// TIA Portal V16 program export: 0 tag tables, 0 data types, 18 data blocks, 36 code blocks (in call order from the OBs), 5 instance data blocks

DATA_BLOCK "dbAlarms"   // DB106
{ S7_Optimized_Access := 'FALSE'; DB_Accessible_From_OPC_UA := 'FALSE' }
VERSION : 0.1
// stored: AutoNumber false, DBAccessibleFromOPCUA false, IsOnlyStoredInLoadMemory false, IsWriteProtectedInAS false
   VAR
      PLI : Array[1..4, 1..32] of Bool;
   END_VAR
BEGIN
   PLI[1,1..32] := FALSE;
   PLI[2,1..32] := FALSE;
   PLI[3,1..32] := FALSE;
   PLI[4,1..32] := FALSE;
END_DATA_BLOCK

DATA_BLOCK "dbDI"   // DB10
{ S7_Optimized_Access := 'FALSE'; DB_Accessible_From_OPC_UA := 'FALSE' }
VERSION : 0.1
// stored: AutoNumber false, DBAccessibleFromOPCUA false, IsOnlyStoredInLoadMemory false, IsWriteProtectedInAS false
   VAR
      ZAUSTAVITEV_V_SILI_NI_AKTIVIRANA : Bool;   // 0=NOT OK, 1=OK
      FOTO_ZAVESA_KANAL_1 : Bool;   // 0=NOT OK, 1=OK
      FOTO_ZAVESA_KANAL_2 : Bool;   // 0=NOT OK, 1=OK
      START_LEVO_NA_VPENJANJU : Bool;
      START_DESNO_NA_VPENJANJU : Bool;
      Spare0_5 : Bool;
      Spare0_6 : Bool;
      PRISOTNOST_ZRAKA_NA_NAPRAVI : Bool;   // 0=NOT OK, 1=OK
      Spare1_0 : Bool;
      Spare1_1 : Bool;
      Spare1_2 : Bool;
      Spare1_3 : Bool;
      Spare1_4 : Bool;
      Spare1_5 : Bool;
      Spare1_6 : Bool;
      Spare1_7 : Bool;
      BIMETAL_TRANSPORTA_NOGIC_IZKLJUCIL : Bool;   // (I0.0) / 0=NOT OK, 1=OK
      VIBRATOR_NOGIC_READY : Bool;   // (I0.1) / 0=NOT READY, 1=READY
      BIMETAL_VIJACENJA_NOGIC_IZKLJUCIL : Bool;   // (I0.2) / 0=NOT OK, 1=OK
      FR_MOTORJA1_ZADAJ_DESNO_READY : Bool;   // (I0.3) / 0=NOT READY, 1=READY
      FR_MOTORJA2_SPREDAJ_DESNO_READY : Bool;   // (I0.4) / 0=NOT READY, 1=READY
      FR_MOTORJA1_ZADAJ_LEVO_READY : Bool;   // (I0.5) / 0=NOT READY, 1=READY
      FR_MOTORJA2_SPREDAJ_LEVO_READY : Bool;   // (I0.6) / 0=NOT READY, 1=READY
      Spare20_7 : Bool;
      FOTOCELICA_TRANSPORTA_NOGIC : Bool;   // (I0.7) / 0=NI PRISOTNO, 1=PRISOTNO | NOT USED
      FOTOCELICA_VSTOP_DRCA_NOGIC : Bool;   // (I1.0) / 0=NI PRISOTNO, 1=PRISOTNO | ? | NOT USED
      FOTOCELICA_PRED_MESTOM_LOCEVANJA : Bool;   // (I1.1) / 0=NI PRISOTNO, 1=PRISOTNO | NOT USED
      FOTOCELICA_VSTOP_DRCA_LEVO : Bool;   // (I1.2) / 0=NI PRISOTNO, 1=PRISOTNO | NOT USED
      FOTOCELICA_VSTOP_DRCA_DESNO : Bool;   // (I1.3) / 0=NI PRISOTNO, 1=PRISOTNO | NOT USED
      FOTOCELICA_LOC_IZH_DRCA_LEVO : Bool;   // (I1.4) / 0=NI PRISOTNO, 1=PRISOTNO | NOT USED
      FOTOCELICA_LOC_IZH_DRCA_DESNO : Bool;   // (I1.5) / 0=NI PRISOTNO, 1=PRISOTNO | NOT USED
      NOGICE_V_VIBRATORJU : Bool;
      ROTACIJSKI_CIL_DESNO : Bool;   // 0=NI PRISOTNO, 1=PRISOTNO
      ROTACIJSKI_CIL_SREDINA : Bool;   // 0=NI PRISOTNO, 1=PRISOTNO
      ROTACIJSKI_CIL_LEVO : Bool;   // 0=NI PRISOTNO, 1=PRISOTNO
      LOC_DRCA_DESNO_NAPREJ : Bool;   // 0=NI PRISOTNO, 1=PRISOTNO | NOT USED
      LOC_DRCA_DESNO_NAZAJ : Bool;   // 0=NI PRISOTNO, 1=PRISOTNO | NOT USED
      LOC_DRCA_LEVO_NAZAJ : Bool;   // 0=NI PRISOTNO, 1=PRISOTNO | NOT USED
      LOC_DRCA_LEVO_NAPREJ : Bool;   // 0=NI PRISOTNO, 1=PRISOTNO | NOT USED
      Spare22_7 : Bool;
      FOTOCELICA_LOC_TRAK_DESNO1 : Bool;   // 0=NI PRISOTNO, 1=PRISOTNO | NOT USED
      FOTOCELICA_LOC_TRAK_DESNO2 : Bool;   // 0=NI PRISOTNO, 1=PRISOTNO | NOT USED
      FOTOCELICA_VIJACENJE_DESNOZADAJ : Bool;   // 0=NI PRISOTNO, 1=PRISOTNO | NOT USED
      FOTOCELICA_VIJACENJE_DESNOSPREDAJ : Bool;   // 0=NI PRISOTNO, 1=PRISOTNO | NOT USED
      VIJACENJE_DESNO_1_NAZAJ : Bool;   // LOCEVANJE NA TRAKU DESNO NAZAJ
      VIJACENJE_DESNO_1_NAPREJ : Bool;   // LOCEVANJE NA TRAKU DESNO NAPREJ
      MESTO_VIJAC_STOP_DESNO_ZAD_NAZAJ : Bool;   // 0=NI PRISOTNO, 1=PRISOTNO
      MESTO_VIJAC_STOP_DESNO_ZAD_NAPREJ : Bool;   // 0=NI PRISOTNO, 1=PRISOTNO
      MESTO_VIJACENJE_DESNO_ZAD_DVIG_DOL : Bool;   // (I1.6) / 0=NI PRISOTNO, 1=PRISOTNO | ? Detekcija spodnje lege cilindra spusta| DONE Man
      MESTO_VIJACENJE_DESNO_ZAD_CENT_NARAZEN : Bool;   // (I1.7) / 0=NI PRISOTNO, 1=PRISOTNO
      MESTO_VIJACENJE_DESNO_ZAD_CENT_SKUPAJ : Bool;   // 0=NI PRISOTNO, 1=PRISOTNO
      Spare24_3 : Bool;   // MESTO_VIJACENJE_DESNO_SPRED_NAZAJ "STOP_DESNO_SPRED_NAZAJ(Spare23_4) ne obstaja. Konec traka ne obstaja cilinder za stopanje nogice.
      Spare24_4 : Bool;   // MESTO_VIJACENJE_DESNO_SPRED_NAPREJ "STOP_DESNO_SPRED_NAPREJ (Spare23_5) ne obstaja. Konec traka ne obstaja cilinder za stopanje nogice.
      MESTO_VIJACENJE_DESNO_SPRED_DVIG_DOL : Bool;   // 0=NI PRISOTNO, 1=PRISOTNO | ? Detekcija spodnje lege cilindra spusta| DONE Man
      MESTO_VIJACENJE_DESNO_SPRED_CENT_NARAZEN : Bool;   // 0=NI PRISOTNO, 1=PRISOTNO
      MESTO_VIJACENJE_DESNO_SPRED_CENT_SKUPAJ : Bool;   // 0=NI PRISOTNO, 1=PRISOTNO
      KONCNA_POZICIJA_VIJACENJA_DES_NAZAJ : Bool;   // 0=NI PRISOTNO, 1=PRISOTNO | NOT USED
      KONCNA_POZICIJA_VIJACENJA_DES_NAPREJ : Bool;   // 0=NI PRISOTNO, 1=PRISOTNO | NOT USED
      Spare25_2 : Bool;
      Spare25_3 : Bool;
      KONCNA_POZICIJA_VIJACENJA_LEVO_NAZAJ : Bool;   // 0=NI PRISOTNO, 1=PRISOTNO | NOT USED
      KONCNA_POZICIJA_VIJACENJA_LEVO_NAPREJ : Bool;   // 0=NI PRISOTNO, 1=PRISOTNO | NOT USED
      Spare25_6 : Bool;
      Spare25_7 : Bool;
      FOTOCELICA_LOC_TRAK_LEVO1 : Bool;   // 0=NI PRISOTNO, 1=PRISOTNO | NOT USED
      FOTOCELICA_LOC_TRAK_LEVO2 : Bool;   // 0=NI PRISOTNO, 1=PRISOTNO | NOT USED
      FOTOCELICA_VIJACENJE_LEVO_ZADAJ : Bool;   // 0=NI PRISOTNO, 1=PRISOTNO | NOT USED
      FOTOCELICA_VIJACENJE_LEVO_SPREDAJ : Bool;   // 0=NI PRISOTNO, 1=PRISOTNO | NOT USED
      VIJACENJE_LEVO_1_NAZAJ : Bool;   // LOCEVANJE NA TRAKU LEVO NAZAJ
      VIJACENJE_LEVO_1_NAPREJ : Bool;   // LOCEVANJE NA TRAKU LEVO NAPREJ
      MESTO_VIJAC_STOP_LEVO_ZAD_NAZAJ : Bool;   // 0=NI PRISOTNO, 1=PRISOTNO
      MESTO_VIJAC_STOP_LEVO_ZAD_NAPREJ : Bool;   // 0=NI PRISOTNO, 1=PRISOTNO
      MESTO_VIJACENJE_LEVO_ZAD_DVIG_DOL : Bool;   // 0=NI PRISOTNO, 1=PRISOTNO | ? Detekcija spodnje lege cilindra spusta| DONE Man
      MESTO_VIJACENJE_LEVO_ZAD_CENT_NARAZEN : Bool;   // 0=NI PRISOTNO, 1=PRISOTNO
      MESTO_VIJACENJE_LEVO_ZAD_CENT_SKUPAJ : Bool;   // 0=NI PRISOTNO, 1=PRISOTNO
      Spare27_3 : Bool;   // MESTO_VIJACENJE_LEVO_SPRED_NAZAJ "STOP_LEVO_SPRED_NAZAJ(Spare26_4) ne obstaja. Konec traka ne obstaja cilinder za stopanje nogice.
      Spare27_4 : Bool;   // MESTO_VIJACENJE_LEVO_SPRED_NAPREJ "STOP_LEVO_SPRED_NAPREJ (Spare26_5) ne obstaja. Konec traka ne obstaja cilinder za stopanje nogice.
      MESTO_VIJACENJE_LEVO_SPRED_DVIG_DOL : Bool;   // 0=NI PRISOTNO, 1=PRISOTNO | ? Detekcija spodnje lege cilindra spusta| DONE Man
      MESTO_VIJACENJE_LEVO_SPRED_CENT_NARAZEN : Bool;   // 0=NI PRISOTNO, 1=PRISOTNO
      MESTO_VIJACENJE_LEVO_SPRED_CENT_SKUPAJ : Bool;   // 0=NI PRISOTNO, 1=PRISOTNO
      INDUKTIVEC_PRAVILNA_VLOZITEV_DNA_1 : Bool;   // 0=NI PRISOTNO, 1=PRISOTNO | NOT USED
      INDUKTIVEC_PRAVILNA_VLOZITEV_DNA_2 : Bool;   // 0=NI PRISOTNO, 1=PRISOTNO | NOT USED
      VPENJANJE_DNA_LEVO_ZADAJ_GOR : Bool;   // 0=NI PRISOTNO, 1=PRISOTNO
      VPENJANJE_DNA_LEVO_ZADAJ_DOL : Bool;   // 0=NI PRISOTNO, 1=PRISOTNO
      VPENJANJE_DNA_LEVO_SPREDAJ_GOR : Bool;   // 0=NI PRISOTNO, 1=PRISOTNO
      VPENJANJE_DNA_LEVO_SPREDAJ_DOL : Bool;   // 0=NI PRISOTNO, 1=PRISOTNO
      VPENJANJE_DNA_DESNO_ZADAJ_GOR : Bool;   // 0=NI PRISOTNO, 1=PRISOTNO
      VPENJANJE_DNA_DESNO_ZADAJ_DOL : Bool;   // 0=NI PRISOTNO, 1=PRISOTNO
      VPENJANJE_DNA_DESNO_SPREDAJ_GOR : Bool;   // 0=NI PRISOTNO, 1=PRISOTNO
      VPENJANJE_DNA_DESNO_SPREDAJ_DOL : Bool;   // 0=NI PRISOTNO, 1=PRISOTNO
      Static_1 : Bool;   // 0=NI PRISOTNO, 1=PRISOTNO
      Spare29_3 : Bool;
      Spare29_4 : Bool;
      Spare29_5 : Bool;
      Spare29_6 : Bool;
      Spare29_7 : Bool;
   END_VAR
BEGIN
END_DATA_BLOCK

DATA_BLOCK "dbDO"   // DB11
{ S7_Optimized_Access := 'FALSE'; DB_Accessible_From_OPC_UA := 'FALSE' }
VERSION : 0.1
// stored: AutoNumber false, DBAccessibleFromOPCUA false, IsOnlyStoredInLoadMemory false, IsWriteProtectedInAS false
   VAR
      SEMAFOR_ZELENA : Bool;
      SEMAFOR_RUMENA : Bool;
      SEMAFOR_RDECA : Bool;
      Spare0_3 { ExternalAccessible := 'False'; ExternalVisible := 'False'; ExternalWritable := 'False'} : Bool;
      Spare0_4 { ExternalAccessible := 'False'; ExternalVisible := 'False'; ExternalWritable := 'False'} : Bool;
      Spare0_5 { ExternalAccessible := 'False'; ExternalVisible := 'False'; ExternalWritable := 'False'} : Bool;
      Spare0_6 { ExternalAccessible := 'False'; ExternalVisible := 'False'; ExternalWritable := 'False'} : Bool;
      Spare0_7 { ExternalAccessible := 'False'; ExternalVisible := 'False'; ExternalWritable := 'False'} : Bool;
      Spare1_0 { ExternalAccessible := 'False'; ExternalVisible := 'False'; ExternalWritable := 'False'} : Bool;
      Spare1_1 { ExternalAccessible := 'False'; ExternalVisible := 'False'; ExternalWritable := 'False'} : Bool;
      Spare1_2 { ExternalAccessible := 'False'; ExternalVisible := 'False'; ExternalWritable := 'False'} : Bool;
      Spare1_3 { ExternalAccessible := 'False'; ExternalVisible := 'False'; ExternalWritable := 'False'} : Bool;
      Spare1_4 { ExternalAccessible := 'False'; ExternalVisible := 'False'; ExternalWritable := 'False'} : Bool;
      Spare1_5 { ExternalAccessible := 'False'; ExternalVisible := 'False'; ExternalWritable := 'False'} : Bool;
      Spare1_6 { ExternalAccessible := 'False'; ExternalVisible := 'False'; ExternalWritable := 'False'} : Bool;
      Spare1_7 { ExternalAccessible := 'False'; ExternalVisible := 'False'; ExternalWritable := 'False'} : Bool;
      VKLOP_M_TRACNEGA_TRANS_NOGIC : Bool;   // (Q0.0)
      VKLOP_VIBRATORJA : Bool;   // (Q0.1)
      VKLOP_M_TRAKA_VIJACNIKA : Bool;   // (Q0.2)
      Spare20_3 { ExternalAccessible := 'False'; ExternalVisible := 'False'; ExternalWritable := 'False'} : Bool;
      Spare20_4 { ExternalAccessible := 'False'; ExternalVisible := 'False'; ExternalWritable := 'False'} : Bool;
      Spare20_5 { ExternalAccessible := 'False'; ExternalVisible := 'False'; ExternalWritable := 'False'} : Bool;
      Spare20_6 { ExternalAccessible := 'False'; ExternalVisible := 'False'; ExternalWritable := 'False'} : Bool;
      Spare20_7 { ExternalAccessible := 'False'; ExternalVisible := 'False'; ExternalWritable := 'False'} : Bool;
      MOTOR_1_ZADAJ_DESNO_START : Bool;   // (Q1.1)
      MOTOR_1_ZADAJ_DESNO_RESET : Bool;   // (Q1.2)
      MOTOR_1_ZADAJ_DESNO_HITROST : Bool;   // (Q1.3)
      MOTOR_1_ZADAJ_DESNO_SMER : Bool;   // (Q1.4)
      MOTOR_2_SPREDAJ_DESNO_START : Bool;   // (Q1.5)
      MOTOR_2_SPREDAJ_DESNO_RESET : Bool;   // (Q1.6)
      MOTOR_2_SPREDAJ_DESNO_HITROST : Bool;   // (Q1.7)
      MOTOR_2_SPREDAJ_DESNO_SMER : Bool;
      MOTOR_1_ZADAJ_LEVO_START : Bool;
      MOTOR_1_ZADAJ_LEVO_RESET : Bool;
      MOTOR_1_ZADAJ_LEVO_HITROST : Bool;
      MOTOR_1_ZADAJ_LEVO_SMER : Bool;
      MOTOR_2_SPREDAJ_LEVO_START : Bool;
      MOTOR_2_SPREDAJ_LEVO_RESET : Bool;
      MOTOR_2_SPREDAJ_LEVO_HITROST : Bool;
      MOTOR_2_SPREDAJ_LEVO_SMER : Bool;
      Spare23_0 { ExternalAccessible := 'False'; ExternalVisible := 'False'; ExternalWritable := 'False'} : Bool;
      Spare23_1 { ExternalAccessible := 'False'; ExternalVisible := 'False'; ExternalWritable := 'False'} : Bool;
      Spare23_2 { ExternalAccessible := 'False'; ExternalVisible := 'False'; ExternalWritable := 'False'} : Bool;
      Spare23_3 { ExternalAccessible := 'False'; ExternalVisible := 'False'; ExternalWritable := 'False'} : Bool;
      Spare23_4 { ExternalAccessible := 'False'; ExternalVisible := 'False'; ExternalWritable := 'False'} : Bool;
      Spare23_5 { ExternalAccessible := 'False'; ExternalVisible := 'False'; ExternalWritable := 'False'} : Bool;
      Spare23_6 { ExternalAccessible := 'False'; ExternalVisible := 'False'; ExternalWritable := 'False'} : Bool;
      Spare23_7 { ExternalAccessible := 'False'; ExternalVisible := 'False'; ExternalWritable := 'False'} : Bool;
   END_VAR
BEGIN
END_DATA_BLOCK

DATA_BLOCK "dbDigitalSensors"   // DB30
{ S7_Optimized_Access := 'FALSE'; DB_Accessible_From_OPC_UA := 'FALSE' }
VERSION : 0.1
// stored: AutoNumber false, DBAccessibleFromOPCUA false, IsOnlyStoredInLoadMemory false, IsWriteProtectedInAS false
   VAR
      ZAUSTAVITEV_V_SILI_NI_AKTIVIRANA : "udtDigitalSensor";
      FOTO_ZAVESA_KANAL_1 : "udtDigitalSensor";
      FOTO_ZAVESA_KANAL_2 : "udtDigitalSensor";
      START_LEVO_NA_VPENJANJU : "udtDigitalSensor";
      START_DESNO_NA_VPENJANJU : "udtDigitalSensor";
      PRISOTNOST_ZRAKA_NA_NAPRAVI : "udtDigitalSensor";
      BIMETAL_TRANSPORTA_NOGIC_IZKLJUCIL : "udtDigitalSensor";
      VIBRATOR_NOGIC_READY : "udtDigitalSensor";
      BIMETAL_VIJACENJA_NOGIC_IZKLJUCIL : "udtDigitalSensor";
      FR_MOTORJA1_ZADAJ_DESNO_READY : "udtDigitalSensor";
      FR_MOTORJA2_SPREDAJ_DESNO_READY : "udtDigitalSensor";
      FR_MOTORJA1_ZADAJ_LEVO_READY : "udtDigitalSensor";
      FR_MOTORJA2_SPREDAJ_LEVO_READY : "udtDigitalSensor";
      Spare20_7 : "udtDigitalSensor";
      FOTOCELICA_TRANSPORTA_NOGIC : "udtDigitalSensor";
      FOTOCELICA_VSTOP_DRCA_NOGIC : "udtDigitalSensor";
      FOTOCELICA_PRED_MESTOM_LOCEVANJA : "udtDigitalSensor";
      FOTOCELICA_VSTOP_DRCA_LEVO : "udtDigitalSensor";
      FOTOCELICA_VSTOP_DRCA_DESNO : "udtDigitalSensor";
      FOTOCELICA_LOC_IZH_DRCA_LEVO : "udtDigitalSensor";
      FOTOCELICA_LOC_IZH_DRCA_DESNO : "udtDigitalSensor";
      NOGICE_V_VIBRATORJU : "udtDigitalSensor";
      ROTACIJSKI_CIL_DESNO : "udtDigitalSensor";
      ROTACIJSKI_CIL_SREDINA : "udtDigitalSensor";
      ROTACIJSKI_CIL_LEVO : "udtDigitalSensor";
      LOC_DRCA_DESNO_NAPREJ : "udtDigitalSensor";
      LOC_DRCA_DESNO_NAZAJ : "udtDigitalSensor";
      LOC_DRCA_LEVO_NAZAJ : "udtDigitalSensor";
      LOC_DRCA_LEVO_NAPREJ : "udtDigitalSensor";
      Spare22_7 : "udtDigitalSensor";
      FOTOCELICA_LOC_TRAK_DESNO1 : "udtDigitalSensor";
      FOTOCELICA_LOC_TRAK_DESNO2 : "udtDigitalSensor";
      FOTOCELICA_VIJACENJE_DESNOZADAJ : "udtDigitalSensor";
      FOTOCELICA_VIJACENJE_DESNOSPREDAJ : "udtDigitalSensor";
      VIJACENJE_DESNO_1_NAZAJ : "udtDigitalSensor";
      VIJACENJE_DESNO_1_NAPREJ : "udtDigitalSensor";
      MESTO_VIJAC_STOP_DESNO_ZAD_NAZAJ : "udtDigitalSensor";
      MESTO_VIJAC_STOP_DESNO_ZAD_NAPREJ : "udtDigitalSensor";
      MESTO_VIJACENJE_DESNO_ZAD_DVIG_DOL : "udtDigitalSensor";
      MESTO_VIJACENJE_DESNO_ZAD_CENT_NARAZEN : "udtDigitalSensor";
      MESTO_VIJACENJE_DESNO_ZAD_CENT_SKUPAJ : "udtDigitalSensor";
      Spare24_3 : "udtDigitalSensor";
      Spare24_4 : "udtDigitalSensor";
      MESTO_VIJACENJE_DESNO_SPRED_DVIG_DOL : "udtDigitalSensor";
      MESTO_VIJACENJE_DESNO_SPRED_CENT_NARAZEN : "udtDigitalSensor";
      MESTO_VIJACENJE_DESNO_SPRED_CENT_SKUPAJ : "udtDigitalSensor";
      KONCNA_POZICIJA_VIJACENJA_DES_NAZAJ : "udtDigitalSensor";
      KONCNA_POZICIJA_VIJACENJA_DES_NAPREJ : "udtDigitalSensor";
      Spare25_2 : "udtDigitalSensor";
      Spare25_3 : "udtDigitalSensor";
      KONCNA_POZICIJA_VIJACENJA_LEVO_NAZAJ : "udtDigitalSensor";
      KONCNA_POZICIJA_VIJACENJA_LEVO_NAPREJ : "udtDigitalSensor";
      Spare25_6 : "udtDigitalSensor";
      Spare25_7 : "udtDigitalSensor";
      FOTOCELICA_LOC_TRAK_LEVO1 : "udtDigitalSensor";
      FOTOCELICA_LOC_TRAK_LEVO2 : "udtDigitalSensor";
      FOTOCELICA_VIJACENJE_LEVO_ZADAJ : "udtDigitalSensor";
      FOTOCELICA_VIJACENJE_LEVO_SPREDAJ : "udtDigitalSensor";
      VIJACENJE_LEVO_1_NAZAJ : "udtDigitalSensor";
      VIJACENJE_LEVO_1_NAPREJ : "udtDigitalSensor";
      MESTO_VIJAC_STOP_LEVO_ZAD_NAZAJ : "udtDigitalSensor";
      MESTO_VIJAC_STOP_LEVO_ZAD_NAPREJ : "udtDigitalSensor";
      MESTO_VIJACENJE_LEVO_ZAD_DVIG_DOL : "udtDigitalSensor";
      MESTO_VIJACENJE_LEVO_ZAD_CENT_NARAZEN : "udtDigitalSensor";
      MESTO_VIJACENJE_LEVO_ZAD_CENT_SKUPAJ : "udtDigitalSensor";
      Spare27_3 : "udtDigitalSensor";
      Spare27_4 : "udtDigitalSensor";
      MESTO_VIJACENJE_LEVO_SPRED_DVIG_DOL : "udtDigitalSensor";
      MESTO_VIJACENJE_LEVO_SPRED_CENT_NARAZEN : "udtDigitalSensor";
      MESTO_VIJACENJE_LEVO_SPRED_CENT_SKUPAJ : "udtDigitalSensor";
      INDUKTIVEC_PRAVILNA_VLOZITEV_DNA_1 : "udtDigitalSensor";
      INDUKTIVEC_PRAVILNA_VLOZITEV_DNA_2 : "udtDigitalSensor";
      VPENJANJE_DNA_LEVO_ZADAJ_GOR : "udtDigitalSensor";
      VPENJANJE_DNA_LEVO_ZADAJ_DOL : "udtDigitalSensor";
      VPENJANJE_DNA_LEVO_SPREDAJ_GOR : "udtDigitalSensor";
      VPENJANJE_DNA_LEVO_SPREDAJ_DOL : "udtDigitalSensor";
      VPENJANJE_DNA_DESNO_ZADAJ_GOR : "udtDigitalSensor";
      VPENJANJE_DNA_DESNO_ZADAJ_DOL : "udtDigitalSensor";
      VPENJANJE_DNA_DESNO_SPREDAJ_GOR : "udtDigitalSensor";
      VPENJANJE_DNA_DESNO_SPREDAJ_DOL : "udtDigitalSensor";
   END_VAR
BEGIN
END_DATA_BLOCK

DATA_BLOCK "dbDigitalValves"   // DB32
{ S7_Optimized_Access := 'FALSE'; DB_Accessible_From_OPC_UA := 'FALSE' }
VERSION : 0.1
// stored: AutoNumber false, DBAccessibleFromOPCUA false, IsOnlyStoredInLoadMemory false, IsWriteProtectedInAS false
   VAR
      Y17_RotCilipozDesno : "udtDigitalValve";   // Crane control not selected lamps (Q0.0)
      Y18_RotCilipozLevo : "udtDigitalValve";
      Y2_VijaDesZad_Dvig : "udtDigitalValve";
      Y3_VijaDesSpr_Dvig : "udtDigitalValve";
      Y4_VijaLevZad_Dvig : "udtDigitalValve";
      Y5_VijaLevSpr_Dvig : "udtDigitalValve";
      Y6_DrcaLocev_Des : "udtDigitalValve";
      Y7_DrcaLocev_Lev : "udtDigitalValve";
      Y8_VijaLocev_Des : "udtDigitalValve";
      Y9_VijaStop_DesZad : "udtDigitalValve";
      Y10_Centri_DesZad : "udtDigitalValve";
      Y11_Centri_DesSpr : "udtDigitalValve";
      Y12_VijaLocev_Lev : "udtDigitalValve";
      Y13_VijaStop_LevZad : "udtDigitalValve";
      Y14_Centri_LevZad : "udtDigitalValve";
      Y15_Centri_LevSpr : "udtDigitalValve";
      Y16_VpenjanjeDna : "udtDigitalValve";
      SEMAFOR_ZELENA : "udtDigitalValve";
      SEMAFOR_RUMENA : "udtDigitalValve";
      SEMAFOR_RDECA : "udtDigitalValve";
   END_VAR
BEGIN
END_DATA_BLOCK

DATA_BLOCK "dbHMIUser"   // DB5
{ S7_Optimized_Access := 'FALSE'; DB_Accessible_From_OPC_UA := 'FALSE' }
VERSION : 0.1
// stored: AutoNumber false, DBAccessibleFromOPCUA false, IsOnlyStoredInLoadMemory false, IsWriteProtectedInAS false
   VAR
      CurrentUsername : String;
      Spare_Bool0 : Bool;
      Spare_2 : Int;
      Spare_3 : Int;
      Spare_4 : UDInt;
      Spare_5 : UDInt;
      Spare_1 : Int;
      SetTargetHMIScreen : Byte;
      HMIScreenJobNo_byte1 : Byte;
      HMIScreenJobNo_byte2 : Byte;
      HMIScreenJobNo_byte3 : Byte;
      HMICurrScreen : Byte;
      HMIScreenJobNo_byte5 : Byte;
      HMIScreenJobNo_byte6 : Byte;
      HMIScreenJobNo_byte7 : Byte;
      HMIScreenJobNo_byte8 : Byte;
      HMIScreenJobNo_byte9 : Byte;
      HMIScreenJobNo_byte10 : Byte;
      HMIScreenJobNo_byte11 : Byte;
      HMIScreenJobNo_byte12 : Byte;
      HMIScreenJobNo_byte13 : Byte;
      HMIScreenJobNo_byte14 : Byte;
      HMIScreenJobNo_byte15 : Byte;
      HMIScreenJobNo_byte16 : Byte;
      HMIScreenJobNo_byte17 : Byte;
      Spare_6 : Int;
      PLCUserLogOut : Int;
      CurrUser_LEN : Int;
      UserLoggOffTime : UDInt := 50;
      CurrMachineStep : String[50];
      HMICurrScreen_OLD { ExternalAccessible := 'False'; ExternalVisible := 'False'; ExternalWritable := 'False'} : Byte;
      PLCUserLogOut_OLD { ExternalAccessible := 'False'; ExternalVisible := 'False'; ExternalWritable := 'False'} : Int;
   END_VAR
BEGIN
END_DATA_BLOCK

DATA_BLOCK "dbHSC"   // DB37
{ S7_Optimized_Access := 'TRUE'; DB_Accessible_From_OPC_UA := 'FALSE' }
VERSION : 0.1
// stored: AutoNumber false, DBAccessibleFromOPCUA false
   VAR RETAIN
      ScanLineCounts { S7_SetPoint := 'True'} : "udtHSC";
   END_VAR
BEGIN
   ScanLineCounts.EguValue := 31.3194;
END_DATA_BLOCK

DATA_BLOCK "dbMotors"   // DB33
{ S7_Optimized_Access := 'TRUE'; DB_Accessible_From_OPC_UA := 'FALSE' }
VERSION : 0.1
// stored: AutoNumber false, DBAccessibleFromOPCUA false, IsOnlyStoredInLoadMemory false, IsRetainMemResEnabled false, IsWriteProtectedInAS false, MemoryReserve 100
   VAR
      VKLOP_M_TRACNEGA_TRANS_NOGIC : "udtMotor";
      M1_ZADAJ_DESNO : "udtMotor";
      M2_SPREDAJ_DESNO : "udtMotor";
      M1_ZADAJ_LEVO : "udtMotor";
      M2_SPREDAJ_LEVO : "udtMotor";
      VKLOP_VIBRATORJA : "udtMotor";
      VKLOP_M_TRAKA_VIJACNIKA : "udtMotor";
   END_VAR
BEGIN
END_DATA_BLOCK

DATA_BLOCK "dbOPAlarms"   // DB112
{ S7_Optimized_Access := 'FALSE'; DB_Accessible_From_OPC_UA := 'FALSE' }
VERSION : 0.1
// stored: AutoNumber false, DBAccessibleFromOPCUA false, IsOnlyStoredInLoadMemory false, IsWriteProtectedInAS false
   VAR
      Alarm : Array[0..63] of Bool;   // System Alarms
      OPAlarmWord : Array[0..3] of Word;   // OP Alarms
      AlarmACK : Array[0..63] of Bool;
   END_VAR
BEGIN
END_DATA_BLOCK

DATA_BLOCK "dbPDO"   // DB12
{ S7_Optimized_Access := 'FALSE'; DB_Accessible_From_OPC_UA := 'FALSE' }
VERSION : 0.1
// stored: AutoNumber false, DBAccessibleFromOPCUA false, IsOnlyStoredInLoadMemory false, IsWriteProtectedInAS false
   VAR
      Spare_00 { ExternalAccessible := 'False'; ExternalVisible := 'False'; ExternalWritable := 'False'} : Bool;
      Spare_01 { ExternalAccessible := 'False'; ExternalVisible := 'False'; ExternalWritable := 'False'} : Bool;
      Y2_VijaDesZad_Dvig { ExternalAccessible := 'False'; ExternalVisible := 'False'; ExternalWritable := 'False'} : Bool;
      Y2_VijaDesZad_Spust { ExternalAccessible := 'False'; ExternalVisible := 'False'; ExternalWritable := 'False'} : Bool;
      Y3_VijaDesSpr_Dvig { ExternalAccessible := 'False'; ExternalVisible := 'False'; ExternalWritable := 'False'} : Bool;
      Y3_VijaDesSpr_Spust { ExternalAccessible := 'False'; ExternalVisible := 'False'; ExternalWritable := 'False'} : Bool;
      Y4_VijaLevZad_Dvig { ExternalAccessible := 'False'; ExternalVisible := 'False'; ExternalWritable := 'False'} : Bool;
      Y4_VijaLevZad_Spust { ExternalAccessible := 'False'; ExternalVisible := 'False'; ExternalWritable := 'False'} : Bool;
      Y5_VijaLevSpr_Dvig { ExternalAccessible := 'False'; ExternalVisible := 'False'; ExternalWritable := 'False'} : Bool;
      Y5_VijaLevSpr_Spust { ExternalAccessible := 'False'; ExternalVisible := 'False'; ExternalWritable := 'False'} : Bool;
      Y6_DrcaLocev_Des { ExternalAccessible := 'False'; ExternalVisible := 'False'; ExternalWritable := 'False'} : Bool;
      Y6_Spare { ExternalAccessible := 'False'; ExternalVisible := 'False'; ExternalWritable := 'False'} : Bool;
      Y7_DrcaLocev_Lev { ExternalAccessible := 'False'; ExternalVisible := 'False'; ExternalWritable := 'False'} : Bool;
      Y7_Spare { ExternalAccessible := 'False'; ExternalVisible := 'False'; ExternalWritable := 'False'} : Bool;
      Y8_VijaLocev_Des { ExternalAccessible := 'False'; ExternalVisible := 'False'; ExternalWritable := 'False'} : Bool;
      Y8_Spare { ExternalAccessible := 'False'; ExternalVisible := 'False'; ExternalWritable := 'False'} : Bool;
      Y9_VijaStop_DesZad { ExternalAccessible := 'False'; ExternalVisible := 'False'; ExternalWritable := 'False'} : Bool;
      Y9_Spare { ExternalAccessible := 'False'; ExternalVisible := 'False'; ExternalWritable := 'False'} : Bool;
      Y10_Centri_DesZad { ExternalAccessible := 'False'; ExternalVisible := 'False'; ExternalWritable := 'False'} : Bool;
      Y10_Spare { ExternalAccessible := 'False'; ExternalVisible := 'False'; ExternalWritable := 'False'} : Bool;
      Y11_Centri_DesSpr { ExternalAccessible := 'False'; ExternalVisible := 'False'; ExternalWritable := 'False'} : Bool;
      Y11_Spare { ExternalAccessible := 'False'; ExternalVisible := 'False'; ExternalWritable := 'False'} : Bool;
      Y12_VijaLocev_Lev { ExternalAccessible := 'False'; ExternalVisible := 'False'; ExternalWritable := 'False'} : Bool;
      Y12_Spare { ExternalAccessible := 'False'; ExternalVisible := 'False'; ExternalWritable := 'False'} : Bool;
      Y13_VijaStop_LevZad { ExternalAccessible := 'False'; ExternalVisible := 'False'; ExternalWritable := 'False'} : Bool;
      Y14_Centri_LevZad { ExternalAccessible := 'False'; ExternalVisible := 'False'; ExternalWritable := 'False'} : Bool;
      Y15_Centri_LevSpr { ExternalAccessible := 'False'; ExternalVisible := 'False'; ExternalWritable := 'False'} : Bool;
      Y16_VpenjanjeDna { ExternalAccessible := 'False'; ExternalVisible := 'False'; ExternalWritable := 'False'} : Bool;
      Y17_RotCilipozDesno { ExternalAccessible := 'False'; ExternalVisible := 'False'; ExternalWritable := 'False'} : Bool;
      Y18_RotCilipozLevo { ExternalAccessible := 'False'; ExternalVisible := 'False'; ExternalWritable := 'False'} : Bool;
   END_VAR
BEGIN
END_DATA_BLOCK

DATA_BLOCK "dbPLCClock"   // DB251
{ S7_Optimized_Access := 'FALSE'; DB_Accessible_From_OPC_UA := 'FALSE' }
VERSION : 0.1
// stored: AutoNumber false, DBAccessibleFromOPCUA false, IsOnlyStoredInLoadMemory false, IsWriteProtectedInAS false
   VAR
      Tenth : Bool := FALSE;
      SEC : Bool := FALSE;
      Minute : Bool := FALSE;
      Hour : Bool := FALSE;
      Day : Bool := FALSE;
      Week : Bool := FALSE;
      Month : Bool := FALSE;
      Year : Bool := FALSE;
      SetPLCClock : Bool := FALSE;
      SetOPPLCClock : Bool := FALSE;
      PLC : "udtClock";
      SCADA : "udtClock";
      SweepTime : Int := 17;
      ScanCounter : Int := 72;
   END_VAR
BEGIN
END_DATA_BLOCK

DATA_BLOCK "dbProfinetAlrm"   // DB4
{ S7_Optimized_Access := 'FALSE'; DB_Accessible_From_OPC_UA := 'FALSE' }
VERSION : 0.0
// stored: AutoNumber true, DBAccessibleFromOPCUA false, IsOnlyStoredInLoadMemory false, IsWriteProtectedInAS false
   VAR
      ProfiNet_Req : Bool := FALSE;
      ProfiNet_SzlID : DWord := 16#0000;
      ProfiNet_Index : Int := 16#0000;
      Profinet_RetVal : Int := 0;
      ProfiNet_Busy : Bool := FALSE;
      ProfiNet_En : Bool := FALSE;
   END_VAR
BEGIN
END_DATA_BLOCK

DATA_BLOCK "dbSystemAlarms"   // DB105
{ S7_Optimized_Access := 'FALSE'; DB_Accessible_From_OPC_UA := 'FALSE' }
VERSION : 0.1
// stored: AutoNumber false, DBAccessibleFromOPCUA false, IsOnlyStoredInLoadMemory false, IsWriteProtectedInAS false
   VAR
      SysAlm : Array[1..1024] of Bool;
      EthAlm : Array[1..128] of Bool;
      DPAlm : Array[1..16, 1..16] of DWord;
   END_VAR
BEGIN
   SysAlm[1..128] := FALSE;
   EthAlm[1..128] := FALSE;
   DPAlm[1,1..16] := 16#0000_0000;
   DPAlm[2,1..16] := 16#0000_0000;
   DPAlm[3,1..16] := 16#0000_0000;
   DPAlm[4,1..16] := 16#0000_0000;
   DPAlm[5,1..16] := 16#0000_0000;
   DPAlm[6,1..16] := 16#0000_0000;
   DPAlm[7,1..16] := 16#0000_0000;
   DPAlm[8,1..16] := 16#0000_0000;
   DPAlm[9,1..16] := 16#0000_0000;
   DPAlm[10,1..16] := 16#0000_0000;
   DPAlm[11,1..16] := 16#0000_0000;
   DPAlm[12,1..16] := 16#0000_0000;
   DPAlm[13,1..16] := 16#0000_0000;
   DPAlm[14,1..16] := 16#0000_0000;
   DPAlm[15,1..16] := 16#0000_0000;
   DPAlm[16,1..16] := 16#0000_0000;
END_DATA_BLOCK

DATA_BLOCK "dbSystemParam"   // DB320
{ S7_Optimized_Access := 'TRUE'; DB_Accessible_From_OPC_UA := 'FALSE' }
VERSION : 0.1
// stored: AutoNumber false, DBAccessibleFromOPCUA false
   VAR RETAIN
      KONCNA_POZICIJA_VIJACENJA_DES_NAZAJ_FilterTime : USInt := 10;
      KONCNA_POZICIJA_VIJACENJA_DES_NAPREJ_FilterTime : USInt := 10;
      KONCNA_POZICIJA_VIJACENJA_LEVO_NAZAJ_FilterTime : USInt := 12;
      KONCNA_POZICIJA_VIJACENJA_LEVO_NAPREJ_FilterTime : USInt := 15;
      DlyTimeToStart_TRAK_VIJAC : Int := 5;
      DlyTimeToStop_TRAK_VIJAC : Int := 1;
      DlyTimeToStart_VIBRO : Int := 5;
      DlyTimeToStop_VIBRO : Int := 15;
      StandbyTimeTrakaVijac : UDInt := 15;
      DlyTimeForAlarmAddNewHelix : UInt := 10;
   END_VAR
BEGIN
END_DATA_BLOCK

DATA_BLOCK "dbTimers"   // DB252
{ S7_Optimized_Access := 'FALSE'; DB_Accessible_From_OPC_UA := 'FALSE' }
VERSION : 0.1
// stored: AutoNumber false, DBAccessibleFromOPCUA false, IsOnlyStoredInLoadMemory false, IsWriteProtectedInAS false
   VAR
      Num : Array[0..40] of "udtTON";
   END_VAR
BEGIN
END_DATA_BLOCK

DATA_BLOCK "dbUnit"   // DB103
{ S7_Optimized_Access := 'FALSE'; DB_Accessible_From_OPC_UA := 'FALSE' }
VERSION : 0.1
// stored: AutoNumber false, DBAccessibleFromOPCUA false, IsOnlyStoredInLoadMemory false, IsWriteProtectedInAS false
   VAR RETAIN
      Unit { S7_SetPoint := 'True'} : Array[1..1] of "udtUnit";
   END_VAR
BEGIN
END_DATA_BLOCK

DATA_BLOCK "dbUtilities"   // DB906
{ S7_Optimized_Access := 'TRUE'; DB_Accessible_From_OPC_UA := 'FALSE' }
VERSION : 0.1
// stored: AutoNumber false, DBAccessibleFromOPCUA false, IsOnlyStoredInLoadMemory false, IsRetainMemResEnabled false, IsWriteProtectedInAS false, MemoryReserve 100
   VAR
      GreenLightFlashFlag : Bool;
      RedLightFlashFlag : Bool;
      BlueLightFlashFlag : Bool;
      YellowLightFlashFlag : Bool;
   END_VAR
BEGIN
END_DATA_BLOCK

DATA_BLOCK "dbWarnings"   // DB107
{ S7_Optimized_Access := 'FALSE'; DB_Accessible_From_OPC_UA := 'FALSE' }
VERSION : 0.1
// stored: AutoNumber false, DBAccessibleFromOPCUA false, IsOnlyStoredInLoadMemory false, IsWriteProtectedInAS false
   VAR
      PLI : Array[1..4, 1..32] of Bool;
   END_VAR
BEGIN
   PLI[1,1..32] := FALSE;
   PLI[2,1..32] := FALSE;
   PLI[3,1..32] := FALSE;
   PLI[4,1..32] := FALSE;
END_DATA_BLOCK

ORGANIZATION_BLOCK "Main"   // OB1, LAD, ProgramCycle
TITLE = "Main Program Sweep (Cycle)"
{ S7_Optimized_Access := 'TRUE' }
VERSION : 0.1
// stored: AutoNumber true, IsIECCheckEnabled false, SetENOAutomatically false
   VAR_INPUT
      Initial_Call : Bool;   // Initial call of this OB
      Remanence : Bool;   // =True, if remanent data are available
   END_VAR
   VAR_TEMP
      OB1_SCAN_1 : Byte;   // 1 (Cold restart scan 1 of OB 1), 3 (Scan 2-n of OB 1)
      OB1_PRIORITY : Byte;   // Priority of OB Execution
      OB1_OB_NUMBR : Byte;   // 1 (Organization block 1, OB1)
      OB1_RESERVED_1 : Byte;   // Reserved for system
      OB1_RESERVED_2 : Byte;   // Reserved for system
      OB1_EV_CLASS : Byte;   // Bits 0-3 = 1 (Coming event), Bits 4-7 = 1 (Event class 1)
      OB1_PREV_CYCLE : Int;   // Cycle time of previous OB1 scan (milliseconds)
      OB1_MIN_CYCLE : Int;   // Minimum cycle time of OB1 (milliseconds)
      OB1_MAX_CYCLE : Int;   // Maximum cycle time of OB1 (milliseconds)
      OB1_DATE_TIME : DTL;   // Date and time OB1 started
   END_VAR
BEGIN

REGION Network 1
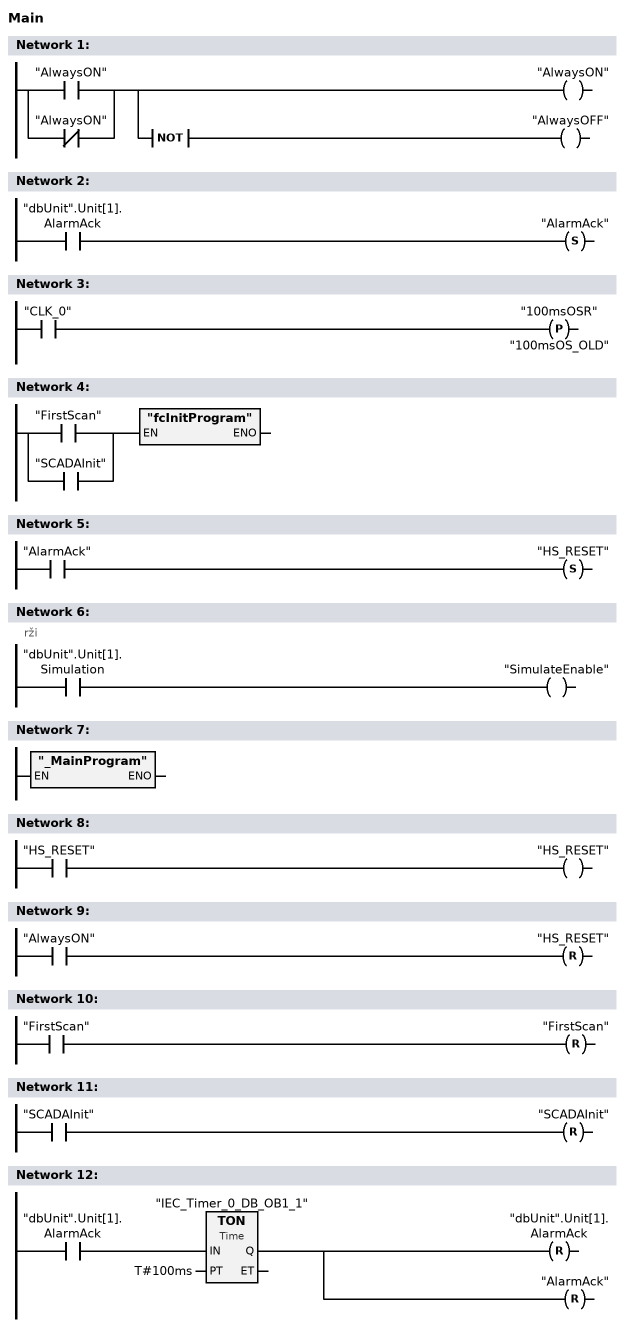
   RUNG wire#powerrail
      Contact( "AlwaysON" )
      wire#w1
      Coil( "AlwaysON" )
   END_RUNG
   RUNG wire#powerrail
      I_Contact( "AlwaysON" )
   END_RUNG wire#w1
   RUNG wire#w1
      Not()
      Coil( "AlwaysOFF" )
   END_RUNG
   // the same network as SCL:
   "AlwaysON" := "AlwaysON" OR NOT "AlwaysON";
   "AlwaysOFF" := NOT "AlwaysON";
END_REGION

REGION Network 2
   RUNG wire#powerrail
      Contact( "dbUnit".Unit[1].AlarmAck )
      S_Coil( "AlarmAck" )
   END_RUNG
   // the same network as SCL:
   IF "dbUnit".Unit[1].AlarmAck THEN "AlarmAck" := TRUE; END_IF;
END_REGION

REGION Network 3
   "100msOSR" := "CLK_0" AND NOT "100msOS_OLD";   // rising edge
   "100msOS_OLD" := "CLK_0";
END_REGION

REGION Network 4
   RUNG wire#powerrail
      Contact( "FirstScan" )
      wire#w1
      "fcInitProgram"()
   END_RUNG
   RUNG wire#powerrail
      Contact( "SCADAInit" )
   END_RUNG wire#w1
   // the same network as SCL:
   IF "FirstScan" OR "SCADAInit" THEN "fcInitProgram"(); END_IF;
END_REGION

REGION Network 5
   RUNG wire#powerrail
      Contact( "AlarmAck" )
      S_Coil( "HS_RESET" )
   END_RUNG
   // the same network as SCL:
   IF "AlarmAck" THEN "HS_RESET" := TRUE; END_IF;
END_REGION

REGION Network 6
   // rži
   RUNG wire#powerrail
      Contact( "dbUnit".Unit[1].Simulation )
      Coil( "SimulateEnable" )
   END_RUNG
   // the same network as SCL:
   "SimulateEnable" := "dbUnit".Unit[1].Simulation;
END_REGION

REGION Network 7
   RUNG wire#powerrail
      "_MainProgram"()
   END_RUNG
   // the same network as SCL:
   "_MainProgram"();
END_REGION

REGION Network 8
   RUNG wire#powerrail
      Contact( "HS_RESET" )
      Coil( "HS_RESET" )
   END_RUNG
   // the same network as SCL:
   "HS_RESET" := "HS_RESET";
END_REGION

REGION Network 9
   RUNG wire#powerrail
      Contact( "AlwaysON" )
      R_Coil( "HS_RESET" )
   END_RUNG
   // the same network as SCL:
   IF "AlwaysON" THEN "HS_RESET" := FALSE; END_IF;
END_REGION

REGION Network 10
   RUNG wire#powerrail
      Contact( "FirstScan" )
      R_Coil( "FirstScan" )
   END_RUNG
   // the same network as SCL:
   IF "FirstScan" THEN "FirstScan" := FALSE; END_IF;
END_REGION

REGION Network 11
   RUNG wire#powerrail
      Contact( "SCADAInit" )
      R_Coil( "SCADAInit" )
   END_RUNG
   // the same network as SCL:
   IF "SCADAInit" THEN "SCADAInit" := FALSE; END_IF;
END_REGION

REGION Network 12
   RUNG wire#powerrail
      Contact( "dbUnit".Unit[1].AlarmAck )
      { S7_Templates := "time_type := Time" } "IEC_Timer_0_DB_OB1_1".TON(pt := T#100ms, et =>)
      wire#w1
      R_Coil( "dbUnit".Unit[1].AlarmAck )
   END_RUNG
   RUNG wire#w1
      R_Coil( "AlarmAck" )
   END_RUNG
   // the same network as SCL:
   "IEC_Timer_0_DB_OB1_1".TON(IN := "dbUnit".Unit[1].AlarmAck, PT := T#100ms);
   IF "IEC_Timer_0_DB_OB1_1".Q THEN
       "dbUnit".Unit[1].AlarmAck := FALSE;
       "AlarmAck" := FALSE;
   END_IF;
END_REGION
END_ORGANIZATION_BLOCK

FUNCTION "fcInitProgram" : Void
{ S7_Optimized_Access := 'FALSE' }
VERSION : 0.1
   VAR_TEMP 
      i : Int;
      DatalogPassedTemp : Bool;
      ErrorTemp : Bool;
      StatusTemp : Word;
      DatalogReq : SInt;
   END_VAR


BEGIN
	// Short summary:
	(*
	  Program initialization
	*)
	// 
	//**********************************************************************
	// Revision control:
	//----------------------------------------------------------------------
	// Use only for revisions of original code
	// V0.01
	// Description of revision
	
	//----------------------------------------------------------------------
	// Comments:
	(*
	  Every change in the code is documented with following:
	  // CCC-yyymmdd: .....
	  yyyy year when change was made
	  mm   month when change was made
	  dd   day when change was made
	  CCC  authors initials
	*)
	//**********************************************************************
	
	//----------------------------------------------------------------------
	// set unit status IDLE
	
	"ProgramMode"               := 0;
	"dbUnit".Unit[1].Regime     := 0;
	"dbUnit".Unit[1].AlarmAck   := True;
	"dbUnit".Unit[1].StartStop  := False;
	
	// init functions
	"fcInitSensors"();
	
	"dbHMIUser".PLCUserLogOut           := 0; // logout current user
	"dbHMIUser".CurrentUsername         := '';
	"dbHMIUser".CurrMachineStep         := 'Naprava resetirana';
	"dbHMIUser".SetTargetHMIScreen      := 0; // Reset activated alarm screen, to prepare for next PLC to HMI screen activation.
	
	"ph_Helix_1_DB".StartCmd            := False;
	"ph_LegsShifter_2_DB".StartCmd      := False;
	"op_ButtonHelix_3_DB".CurrentStep   := 0;
	
END_FUNCTION

FUNCTION "fcInitSensors" : Void
{ S7_Optimized_Access := 'FALSE' }
VERSION : 0.1

BEGIN
	// Short summary:
	(*
	  Initialization of sensors
	*)
	// 
	//**********************************************************************
	// Revision control:
	//----------------------------------------------------------------------
	// Use only for revisions of original code
	// V0.01
	// Description of revision
	
	//----------------------------------------------------------------------
	// Comments:
	(*
	  Every change in the code is documented with following:
	  // CCC-yyymmdd: .....
	  yyyy year when change was made
	  mm   month when change was made
	  dd   day when change was made
	  CCC  authors initials
	*)
	//**********************************************************************
	
	//----------------------------------------------------------------------
	//  Digital Sensors
	// Invert
	// CPU Inputs
	"dbDigitalSensors".ZAUSTAVITEV_V_SILI_NI_AKTIVIRANA.Invert  := False;
	"dbDigitalSensors".FOTO_ZAVESA_KANAL_1.Invert               := False;
	"dbDigitalSensors".FOTO_ZAVESA_KANAL_2.Invert               := False;
	"dbDigitalSensors".START_LEVO_NA_VPENJANJU.Invert           := False;
	"dbDigitalSensors".START_DESNO_NA_VPENJANJU.Invert          := False;
	"dbDigitalSensors".PRISOTNOST_ZRAKA_NA_NAPRAVI.Invert       := False;
	// Weidmuller inputs
	"dbDigitalSensors".BIMETAL_TRANSPORTA_NOGIC_IZKLJUCIL.Invert  := False;
	"dbDigitalSensors".VIBRATOR_NOGIC_READY.Invert                := False;
	"dbDigitalSensors".BIMETAL_VIJACENJA_NOGIC_IZKLJUCIL.Invert   := False;
	"dbDigitalSensors".FR_MOTORJA1_ZADAJ_DESNO_READY.Invert       := False;
	"dbDigitalSensors".FR_MOTORJA2_SPREDAJ_DESNO_READY.Invert     := False;
	"dbDigitalSensors".FR_MOTORJA1_ZADAJ_LEVO_READY.Invert        := False;
	"dbDigitalSensors".FR_MOTORJA2_SPREDAJ_LEVO_READY.Invert      := False;
	"dbDigitalSensors".Spare20_7.Invert                           := False;
	"dbDigitalSensors".FOTOCELICA_TRANSPORTA_NOGIC.Invert         := False;
	"dbDigitalSensors".FOTOCELICA_VSTOP_DRCA_NOGIC.Invert         := False;
	"dbDigitalSensors".FOTOCELICA_PRED_MESTOM_LOCEVANJA.Invert    := False;
	"dbDigitalSensors".FOTOCELICA_VSTOP_DRCA_LEVO.Invert          := False;
	"dbDigitalSensors".FOTOCELICA_VSTOP_DRCA_DESNO.Invert         := False;
	"dbDigitalSensors".FOTOCELICA_LOC_IZH_DRCA_LEVO.Invert        := False;
	"dbDigitalSensors".FOTOCELICA_LOC_IZH_DRCA_DESNO.Invert       := False;
	"dbDigitalSensors".NOGICE_V_VIBRATORJU.Invert                 := False;
	"dbDigitalSensors".ROTACIJSKI_CIL_DESNO.Invert                := False;
	"dbDigitalSensors".ROTACIJSKI_CIL_SREDINA.Invert              := False;
	"dbDigitalSensors".ROTACIJSKI_CIL_LEVO.Invert                 := False;
	"dbDigitalSensors".LOC_DRCA_DESNO_NAPREJ.Invert               := False;
	"dbDigitalSensors".LOC_DRCA_DESNO_NAZAJ.Invert                := False;
	"dbDigitalSensors".LOC_DRCA_LEVO_NAZAJ.Invert                 := False;
	"dbDigitalSensors".LOC_DRCA_LEVO_NAPREJ.Invert                := False;
	"dbDigitalSensors".Spare22_7.Invert                           := False;
	"dbDigitalSensors".FOTOCELICA_LOC_TRAK_DESNO1.Invert          := False;
	"dbDigitalSensors".FOTOCELICA_LOC_TRAK_DESNO2.Invert          := False;
	"dbDigitalSensors".FOTOCELICA_VIJACENJE_DESNOZADAJ.Invert     := False;
	"dbDigitalSensors".FOTOCELICA_VIJACENJE_DESNOSPREDAJ.Invert   := False;
	"dbDigitalSensors".VIJACENJE_DESNO_1_NAZAJ.Invert             := False;
	"dbDigitalSensors".VIJACENJE_DESNO_1_NAPREJ.Invert            := False;
	"dbDigitalSensors".MESTO_VIJAC_STOP_DESNO_ZAD_NAZAJ.Invert    := False;
	"dbDigitalSensors".MESTO_VIJAC_STOP_DESNO_ZAD_NAPREJ.Invert   := False;
	"dbDigitalSensors".MESTO_VIJACENJE_DESNO_ZAD_DVIG_DOL.Invert  := False;
	"dbDigitalSensors".MESTO_VIJACENJE_DESNO_ZAD_CENT_NARAZEN.Invert  := False;
	"dbDigitalSensors".MESTO_VIJACENJE_DESNO_ZAD_CENT_SKUPAJ.Invert   := False;
	"dbDigitalSensors".Spare24_3.Invert                               := False;
	"dbDigitalSensors".Spare24_4.Invert                               := False;
	"dbDigitalSensors".MESTO_VIJACENJE_DESNO_SPRED_DVIG_DOL.Invert      := False;
	"dbDigitalSensors".MESTO_VIJACENJE_DESNO_SPRED_CENT_NARAZEN.Invert  := False;
	"dbDigitalSensors".MESTO_VIJACENJE_DESNO_SPRED_CENT_SKUPAJ.Invert   := False;
	"dbDigitalSensors".KONCNA_POZICIJA_VIJACENJA_DES_NAZAJ.Invert       := False;
	"dbDigitalSensors".KONCNA_POZICIJA_VIJACENJA_DES_NAPREJ.Invert      := False;
	"dbDigitalSensors".Spare25_2.Invert                                 := False;
	"dbDigitalSensors".Spare25_3.Invert                                 := False;
	"dbDigitalSensors".KONCNA_POZICIJA_VIJACENJA_LEVO_NAZAJ.Invert      := False;
	"dbDigitalSensors".KONCNA_POZICIJA_VIJACENJA_LEVO_NAPREJ.Invert     := False;
	"dbDigitalSensors".Spare25_6.Invert                                 := False;
	"dbDigitalSensors".Spare25_7.Invert                                 := False;
	"dbDigitalSensors".FOTOCELICA_LOC_TRAK_LEVO1.Invert                 := False;
	"dbDigitalSensors".FOTOCELICA_LOC_TRAK_LEVO2.Invert                 := False;
	"dbDigitalSensors".FOTOCELICA_VIJACENJE_LEVO_ZADAJ.Invert           := False;
	"dbDigitalSensors".FOTOCELICA_VIJACENJE_LEVO_SPREDAJ.Invert         := False;
	"dbDigitalSensors".VIJACENJE_LEVO_1_NAZAJ.Invert                    := False;
	"dbDigitalSensors".VIJACENJE_LEVO_1_NAPREJ.Invert                   := False;
	"dbDigitalSensors".MESTO_VIJAC_STOP_LEVO_ZAD_NAZAJ.Invert           := False;
	"dbDigitalSensors".MESTO_VIJAC_STOP_LEVO_ZAD_NAPREJ.Invert          := False;
	"dbDigitalSensors".MESTO_VIJACENJE_LEVO_ZAD_DVIG_DOL.Invert         := False;
	"dbDigitalSensors".MESTO_VIJACENJE_LEVO_ZAD_CENT_NARAZEN.Invert     := False;
	"dbDigitalSensors".MESTO_VIJACENJE_LEVO_ZAD_CENT_SKUPAJ.Invert      := False;
	"dbDigitalSensors".Spare27_3.Invert                                 := False;
	"dbDigitalSensors".Spare27_4.Invert                                 := False;
	"dbDigitalSensors".MESTO_VIJACENJE_LEVO_SPRED_DVIG_DOL.Invert       := False;
	"dbDigitalSensors".MESTO_VIJACENJE_LEVO_SPRED_CENT_NARAZEN.Invert   := False;
	"dbDigitalSensors".MESTO_VIJACENJE_LEVO_SPRED_CENT_SKUPAJ.Invert    := False;
	"dbDigitalSensors".INDUKTIVEC_PRAVILNA_VLOZITEV_DNA_1.Invert        := False;
	"dbDigitalSensors".INDUKTIVEC_PRAVILNA_VLOZITEV_DNA_2.Invert        := False;
	"dbDigitalSensors".VPENJANJE_DNA_LEVO_ZADAJ_GOR.Invert              := False;
	"dbDigitalSensors".VPENJANJE_DNA_LEVO_ZADAJ_DOL.Invert              := False;
	"dbDigitalSensors".VPENJANJE_DNA_LEVO_SPREDAJ_GOR.Invert            := False;
	"dbDigitalSensors".VPENJANJE_DNA_LEVO_SPREDAJ_DOL.Invert            := False;
	"dbDigitalSensors".VPENJANJE_DNA_DESNO_ZADAJ_GOR.Invert             := False;
	"dbDigitalSensors".VPENJANJE_DNA_DESNO_ZADAJ_DOL.Invert             := False;
	"dbDigitalSensors".VPENJANJE_DNA_DESNO_SPREDAJ_GOR.Invert           := False;
	"dbDigitalSensors".VPENJANJE_DNA_DESNO_SPREDAJ_DOL.Invert           := False;
	"dbDigitalSensors".NOGICE_V_VIBRATORJU.Invert                       := False;
	
	// FilterTime
	"dbDigitalSensors".ZAUSTAVITEV_V_SILI_NI_AKTIVIRANA.FilterTime          := 0;
	"dbDigitalSensors".FOTO_ZAVESA_KANAL_1.FilterTime                       := 0;
	"dbDigitalSensors".FOTO_ZAVESA_KANAL_2.FilterTime                       := 0;
	"dbDigitalSensors".START_LEVO_NA_VPENJANJU.FilterTime                   := 1;
	"dbDigitalSensors".START_DESNO_NA_VPENJANJU.FilterTime                  := 1;
	"dbDigitalSensors".PRISOTNOST_ZRAKA_NA_NAPRAVI.FilterTime               := 0;
	"dbDigitalSensors".BIMETAL_VIJACENJA_NOGIC_IZKLJUCIL.FilterTime         := 0;
	"dbDigitalSensors".VIBRATOR_NOGIC_READY.FilterTime                      := 0;
	"dbDigitalSensors".BIMETAL_VIJACENJA_NOGIC_IZKLJUCIL.FilterTime         := 0;
	"dbDigitalSensors".FR_MOTORJA1_ZADAJ_DESNO_READY.FilterTime             := 0;
	"dbDigitalSensors".FR_MOTORJA2_SPREDAJ_DESNO_READY.FilterTime           := 0;
	"dbDigitalSensors".FR_MOTORJA1_ZADAJ_LEVO_READY.FilterTime              := 0;
	"dbDigitalSensors".FR_MOTORJA2_SPREDAJ_LEVO_READY.FilterTime            := 0;
	"dbDigitalSensors".Spare20_7.FilterTime                                 := 0;
	"dbDigitalSensors".FOTOCELICA_TRANSPORTA_NOGIC.FilterTime               := 30;
	"dbDigitalSensors".FOTOCELICA_VSTOP_DRCA_NOGIC.FilterTime               := 5;
	"dbDigitalSensors".FOTOCELICA_PRED_MESTOM_LOCEVANJA.FilterTime          := 5;
	"dbDigitalSensors".FOTOCELICA_VSTOP_DRCA_LEVO.FilterTime                := 10; // Delect helix only when line is full, helix flying through must NOT be detected
	"dbDigitalSensors".FOTOCELICA_VSTOP_DRCA_DESNO.FilterTime               := 10; // Delect helix only when line is full, helix flying through must NOT be detected
	"dbDigitalSensors".FOTOCELICA_LOC_IZH_DRCA_LEVO.FilterTime              := 5;
	"dbDigitalSensors".FOTOCELICA_LOC_IZH_DRCA_DESNO.FilterTime             := 5;
	"dbDigitalSensors".NOGICE_V_VIBRATORJU.FilterTime                       := 0;
	"dbDigitalSensors".ROTACIJSKI_CIL_DESNO.FilterTime                      := 3;
	"dbDigitalSensors".ROTACIJSKI_CIL_SREDINA.FilterTime                    := 3;
	"dbDigitalSensors".ROTACIJSKI_CIL_LEVO.FilterTime                       := 3;
	"dbDigitalSensors".LOC_DRCA_DESNO_NAPREJ.FilterTime                     := 3;
	"dbDigitalSensors".LOC_DRCA_DESNO_NAZAJ.FilterTime                      := 3;
	"dbDigitalSensors".LOC_DRCA_LEVO_NAZAJ.FilterTime                       := 3;
	"dbDigitalSensors".LOC_DRCA_LEVO_NAPREJ.FilterTime                      := 3;
	"dbDigitalSensors".Spare22_7.FilterTime                                 := 0;
	"dbDigitalSensors".FOTOCELICA_LOC_TRAK_DESNO1.FilterTime                := 0;
	"dbDigitalSensors".FOTOCELICA_LOC_TRAK_DESNO2.FilterTime                := 0;
	"dbDigitalSensors".FOTOCELICA_VIJACENJE_DESNOZADAJ.FilterTime           := 10;
	"dbDigitalSensors".FOTOCELICA_VIJACENJE_DESNOSPREDAJ.FilterTime         := 10;
	"dbDigitalSensors".VIJACENJE_DESNO_1_NAZAJ.FilterTime                   := 3;
	"dbDigitalSensors".VIJACENJE_DESNO_1_NAPREJ.FilterTime                  := 3;
	"dbDigitalSensors".MESTO_VIJAC_STOP_DESNO_ZAD_NAZAJ.FilterTime          := 3;
	"dbDigitalSensors".MESTO_VIJAC_STOP_DESNO_ZAD_NAPREJ.FilterTime         := 3;
	"dbDigitalSensors".MESTO_VIJACENJE_DESNO_ZAD_DVIG_DOL.FilterTime        := 15;
	"dbDigitalSensors".MESTO_VIJACENJE_DESNO_ZAD_CENT_NARAZEN.FilterTime    := 3;
	"dbDigitalSensors".MESTO_VIJACENJE_DESNO_ZAD_CENT_SKUPAJ.FilterTime     := 3;
	"dbDigitalSensors".Spare24_3.FilterTime                                 := 3;
	"dbDigitalSensors".Spare24_4.FilterTime                                 := 3;
	"dbDigitalSensors".MESTO_VIJACENJE_DESNO_SPRED_DVIG_DOL.FilterTime      := 15;
	"dbDigitalSensors".MESTO_VIJACENJE_DESNO_SPRED_CENT_NARAZEN.FilterTime  := 3;
	"dbDigitalSensors".MESTO_VIJACENJE_DESNO_SPRED_CENT_SKUPAJ.FilterTime   := 3;
	// "dbDigitalSensors".KONCNA_POZICIJA_VIJACENJA_DES_NAZAJ.FilterTime       := "dbSystemParam".KONCNA_POZICIJA_VIJACENJA_DES_NAZAJ_FilterTime;  // Moved to fcUtilities
	// "dbDigitalSensors".KONCNA_POZICIJA_VIJACENJA_DES_NAPREJ.FilterTime      := "dbSystemParam".KONCNA_POZICIJA_VIJACENJA_DES_NAPREJ_FilterTime; // Moved to fcUtilities
	"dbDigitalSensors".Spare25_2.FilterTime                                 := 0;
	"dbDigitalSensors".Spare25_3.FilterTime                                 := 0;
	// "dbDigitalSensors".KONCNA_POZICIJA_VIJACENJA_LEVO_NAZAJ.FilterTime      := "dbSystemParam".KONCNA_POZICIJA_VIJACENJA_LEVO_NAZAJ_FilterTime; // Moved to fcUtilities
	// "dbDigitalSensors".KONCNA_POZICIJA_VIJACENJA_LEVO_NAPREJ.FilterTime     := "dbSystemParam".KONCNA_POZICIJA_VIJACENJA_DES_NAPREJ_FilterTime; // Moved to fcUtilities
	"dbDigitalSensors".Spare25_6.FilterTime                                 := 0;
	"dbDigitalSensors".Spare25_7.FilterTime                                 := 0;
	"dbDigitalSensors".FOTOCELICA_LOC_TRAK_LEVO1.FilterTime                 := 0;
	"dbDigitalSensors".FOTOCELICA_LOC_TRAK_LEVO2.FilterTime                 := 0;
	"dbDigitalSensors".FOTOCELICA_VIJACENJE_LEVO_ZADAJ.FilterTime           := 10;
	"dbDigitalSensors".FOTOCELICA_VIJACENJE_LEVO_SPREDAJ.FilterTime         := 10;
	"dbDigitalSensors".VIJACENJE_LEVO_1_NAZAJ.FilterTime                    := 3;
	"dbDigitalSensors".VIJACENJE_LEVO_1_NAPREJ.FilterTime                   := 3;
	"dbDigitalSensors".MESTO_VIJAC_STOP_LEVO_ZAD_NAZAJ.FilterTime           := 3;
	"dbDigitalSensors".MESTO_VIJAC_STOP_LEVO_ZAD_NAPREJ.FilterTime          := 3;
	"dbDigitalSensors".MESTO_VIJACENJE_LEVO_ZAD_DVIG_DOL.FilterTime         := 15;
	"dbDigitalSensors".MESTO_VIJACENJE_LEVO_ZAD_CENT_NARAZEN.FilterTime     := 3;
	"dbDigitalSensors".MESTO_VIJACENJE_LEVO_ZAD_CENT_SKUPAJ.FilterTime      := 3;
	"dbDigitalSensors".Spare27_3.FilterTime                                 := 3;
	"dbDigitalSensors".Spare27_4.FilterTime                                 := 3;
	"dbDigitalSensors".MESTO_VIJACENJE_LEVO_SPRED_DVIG_DOL.FilterTime       := 15;
	"dbDigitalSensors".MESTO_VIJACENJE_LEVO_SPRED_CENT_NARAZEN.FilterTime   := 3;
	"dbDigitalSensors".MESTO_VIJACENJE_LEVO_SPRED_CENT_SKUPAJ.FilterTime    := 3;
	"dbDigitalSensors".INDUKTIVEC_PRAVILNA_VLOZITEV_DNA_1.FilterTime        := 3;
	"dbDigitalSensors".INDUKTIVEC_PRAVILNA_VLOZITEV_DNA_2.FilterTime        := 3;
	"dbDigitalSensors".VPENJANJE_DNA_LEVO_ZADAJ_GOR.FilterTime              := 3;
	"dbDigitalSensors".VPENJANJE_DNA_LEVO_ZADAJ_DOL.FilterTime              := 3;
	"dbDigitalSensors".VPENJANJE_DNA_LEVO_SPREDAJ_GOR.FilterTime            := 3;
	"dbDigitalSensors".VPENJANJE_DNA_LEVO_SPREDAJ_DOL.FilterTime            := 3;
	"dbDigitalSensors".VPENJANJE_DNA_DESNO_ZADAJ_GOR.FilterTime             := 3;
	"dbDigitalSensors".VPENJANJE_DNA_DESNO_ZADAJ_DOL.FilterTime             := 3;
	"dbDigitalSensors".VPENJANJE_DNA_DESNO_SPREDAJ_GOR.FilterTime           := 3;
	"dbDigitalSensors".VPENJANJE_DNA_DESNO_SPREDAJ_DOL.FilterTime           := 3;
END_FUNCTION

FUNCTION "_MainProgram" : Void
{ S7_Optimized_Access := 'FALSE' }
VERSION : 0.1
   VAR_TEMP 
      tmpINT : Int;
      k : Int;
   END_VAR


BEGIN
	//**********************************************************************
	// Project:      P21003
	// Source name:  _MainProgram
	// Author:       PRA: R-TRONIC Slovenia-EU
	// Date:         20210322
	// Version:      0.01
	// Reference:    Vijacenje nog v dno pečice MiniTec, d.o.o.
	//**********************************************************************
	// Short summary:
	(*
	  Main PLC program
	*)
	// 
	//**********************************************************************
	// Revision control:
	//----------------------------------------------------------------------
	// Use only for revisions of original code
	// V0.01
	// Description of revision
	
	//----------------------------------------------------------------------
	// Comments:
	(*
	  Every change in the code is documented with following:
	  // CCC-yyymmdd: .....
	  yyyy year when change was made
	  mm   month when change was made
	  dd   day when change was made
	  CCC  authors initials
	*)
	//**********************************************************************
	
	"SWVersion" := 2.00;
	
	//======================================================================
	//                           Main Program                              //
	//======================================================================
	//----------------------------------------------------------------------
	//  INIT Global Variables
	"MaxPLITimersIndex" := 4;
	
	//  ProgramMode (MW2) = 0=normal, 1=IQ, 2=Simulation
	IF ("ProgramMode" < 0 OR "ProgramMode" > 2) THEN "ProgramMode" := 0; END_IF;
	
	//================================ READ ================================
	//  Ignore if ProgramMode is set to Simulation
	IF "ProgramMode" <> 2 THEN "fcReadIN"(); END_IF;
	
	//================================ RUN =================================
	//  Ignore if ProgramMode is set to IQ
	IF "ProgramMode" <> 1 THEN
	//----------------------------------------------------------------------
	//  Global functions
	   // PRA "PLC_CLOCK"();           //  PLC clock
	    // To se stestiram in dost za danes
	    // To se stestiram in dost za danes 2
	    
	//----------------------------------------------------------------------
	//  Control Modules - inputs
	  "fcDigitalSensors"();    //  Digital Sensors
	  "fcHSCEncoder"();
	
	//----------------------------------------------------------------------
	//  System functions
	  "fcSystemAlarms"();      //  System Alarms
	  "fcResetAvto"();         //  Reset Avto Commands
	  "fcOPAlarming"();        //  Generate HMI alarms
	  
	//----------------------------------------------------------------------
	//  UNIT SUPERVISON
	  "fcUnitInterlocks"();    //  Unit interlocks
	
	//  Procedural Model
	  "TIMER_ON_DELAY"();      //  PLI Timers  
	  "fcImplementation"();
	   
	// Utilities   
	   "fcUtilities"();         //  Program utilities
	   
	//----------------------------------------------------------------------
	//  Control Modules - outputs
	   "fcDigitalValves"();     //  Digital on/off elements
	   "fcMotors"();            //  Motors elements
	   
	END_IF;
	
	//=============================== WRITE ================================
	//  Ignore if ProgramMode is set to Simulation
	IF "ProgramMode" <> 2 THEN "fcWriteOUT"(); END_IF;
END_FUNCTION

FUNCTION "fcReadIN" : Void
{ S7_Optimized_Access := 'TRUE' }
VERSION : 0.1

BEGIN
	// Read DI input (14x) from CPU
	// Read input from I0.0-I1.0 with 2 bytes to DB10.DBB0
	POKE_BLK(area_src:=16#81, // PI
	         dbNumber_src:=0,
	         byteOffset_src:=0,
	         area_dest:=16#84, // DB
	         dbNumber_dest:=10,
	         byteOffset_dest:=0,
	         count:=2);
	
	// Read DI input (16x5) from Weidmuller UR20-FBC-PN-IRT-V2
	// Read input from I2.0-I11.0 with 10 bytes to DB10.DBB2
	POKE_BLK(area_src := 16#81, // PI
	         dbNumber_src := 0,
	         byteOffset_src := 2,
	         area_dest := 16#84, // DB
	         dbNumber_dest := 10,
	         byteOffset_dest := 2,
	         count := 10);
	
END_FUNCTION

FUNCTION "PLC_CLOCK" : Void
{ S7_Optimized_Access := 'FALSE' }
VERSION : 0.1
   VAR_TEMP 
      DANDT {InstructionName := 'DTL'; LibVersion := '1.0'} : DTL;
      DANDT1 : Time;
      word_temp : Word;
      DINT_TEMP : DInt;
      Error : Int;
   END_VAR


BEGIN
	//-------------------- Sweep Time --------------------
	#Error := RD_LOC_T(OUT => #DANDT);
	#DANDT1 := T_DIFF(IN1 := #DANDT, IN2 := "dbPLCClock".PLC.CurrentDateAndTime); // TIME
	#DINT_TEMP := TIME_TO_DINT(#DANDT1);
	
	IF DINT_TO_INT(#DINT_TEMP) >= 0 THEN
	    "dbPLCClock".SweepTime := DINT_TO_INT(#DINT_TEMP);
	ELSIF DINT_TO_INT(#DINT_TEMP) < 0 THEN
	    "dbPLCClock".SweepTime := "dbPLCClock".SweepTime;
	END_IF;
	"dbPLCClock".PLC.CurrentDateAndTime := #DANDT; //
	
	//-------------------- YEAR ---------------------------------------------
	"dbPLCClock".Year := FALSE;
	
	IF "dbPLCClock".PLC.CurrentYear <> "dbPLCClock".PLC.CurrentDateAndTime.YEAR THEN
	    "dbPLCClock".Year := TRUE;
	END_IF;
	"dbPLCClock".PLC.CurrentYear := "dbPLCClock".PLC.CurrentDateAndTime.YEAR;
	
	//------------------------ MONTH ------------------------------------------
	"dbPLCClock".Month := FALSE;
	
	IF "dbPLCClock".PLC.CurrentMonth <> "dbPLCClock".PLC.CurrentDateAndTime.MONTH THEN
	    "dbPLCClock".Month := TRUE;
	END_IF;
	"dbPLCClock".PLC.CurrentMonth := "dbPLCClock".PLC.CurrentDateAndTime.MONTH;
	
	//-------------------- DAY ---------------------------------------------
	"dbPLCClock".Day := FALSE;
	
	IF "dbPLCClock".PLC.CurrentDayOfMonth <> "dbPLCClock".PLC.CurrentDateAndTime.DAY THEN
	    "dbPLCClock".Day := TRUE;
	END_IF;
	"dbPLCClock".PLC.CurrentDayOfMonth := "dbPLCClock".PLC.CurrentDateAndTime.DAY;
	
	//------------------- HOUR --------------------------------------------------
	"dbPLCClock".Hour := FALSE;
	
	IF "dbPLCClock".PLC.CurrentHour <> "dbPLCClock".PLC.CurrentDateAndTime.HOUR THEN
	    "dbPLCClock".Hour := TRUE;
	END_IF;
	"dbPLCClock".PLC.CurrentHour := "dbPLCClock".PLC.CurrentDateAndTime.HOUR;
	
	//-------------------- MINUTE---------------------------------------------
	"dbPLCClock".Minute := FALSE;
	
	IF "dbPLCClock".PLC.CurrentMinute <> "dbPLCClock".PLC.CurrentDateAndTime.MINUTE THEN
	    "dbPLCClock".Minute := TRUE;
	END_IF;
	"dbPLCClock".PLC.CurrentMinute := "dbPLCClock".PLC.CurrentDateAndTime.MINUTE;
	
	//------------------- SECOND---------------------------------------------
	"dbPLCClock".SEC := FALSE;
	
	IF "dbPLCClock".PLC.CurrentSecond <> "dbPLCClock".PLC.CurrentDateAndTime.SECOND THEN
	    "dbPLCClock".SEC := TRUE;
	END_IF;
	"dbPLCClock".PLC.CurrentSecond := "dbPLCClock".PLC.CurrentDateAndTime.SECOND;
	
	//------------------- CURRENT DAY ---------------------------------------------
	// PON = 1; Siemens format: NED = 1
	"dbPLCClock".PLC.CurrentDay := "dbPLCClock".PLC.CurrentDateAndTime.WEEKDAY;
	"dbPLCClock".PLC.CurrentDay := "dbPLCClock".PLC.CurrentDay - 1;
	IF "dbPLCClock".PLC.CurrentDay = -1 THEN
	    "dbPLCClock".PLC.CurrentDay := 7; // Sunday
	END_IF;
	
	// global variables
	"SekOSR" := "dbPLCClock".SEC;
	"MinOSR" := "dbPLCClock".Minute;
	"HourOSR" := "dbPLCClock".Hour;
	"DayOSR" := "dbPLCClock".Day;
	"MonthOSR" := "dbPLCClock".Month;
	"YearOSR" := "dbPLCClock".Year;
	
	//---------------------- Set PLC clock ----------------------
	IF "dbPLCClock".SetPLCClock THEN
	    "dbPLCClock".SetPLCClock := FALSE;
	    #Error := WR_SYS_T(IN := "dbPLCClock".SCADA.CurrentDateAndTime);
	END_IF;
	
	//---------------------- WatchDog Data for PDM ----------------------
	"dbPLCClock".ScanCounter := "dbPLCClock".PLC.CurrentSecond;
	
END_FUNCTION

FUNCTION "fcDigitalSensors" : Void
{ S7_Optimized_Access := 'FALSE' }
VERSION : 0.1
   VAR_TEMP 
      Simulate : Int;
   END_VAR


BEGIN
	// Short summary:
	(*
	  Digital sensors input read and function call
	*)
	// 
	//**********************************************************************
	// Revision control:
	//----------------------------------------------------------------------
	// Use only for revisions of original code
	// V0.01
	// Description of revision
	
	//----------------------------------------------------------------------
	// Comments:
	(*
	  Every change in the code is documented with following:
	  // CCC-yyymmdd: .....
	  yyyy year when change was made
	  mm   month when change was made
	  dd   day when change was made
	  CCC  authors initials
	*)
	//**********************************************************************
	
	// update simulate enable signal
	IF "SimulateEnable" THEN
	  #Simulate := 1;
	ELSE
	  #Simulate := 0;
	END_IF;
	
	//----------------------------------------------------------------------
	//  read input
	"dbDigitalSensors".ZAUSTAVITEV_V_SILI_NI_AKTIVIRANA.Input           := "dbDI".ZAUSTAVITEV_V_SILI_NI_AKTIVIRANA;
	"dbDigitalSensors".FOTO_ZAVESA_KANAL_1.Input                        := "dbDI".FOTO_ZAVESA_KANAL_1;
	"dbDigitalSensors".FOTO_ZAVESA_KANAL_2.Input                        := "dbDI".FOTO_ZAVESA_KANAL_2;
	"dbDigitalSensors".START_LEVO_NA_VPENJANJU.Input                    := "dbDI".START_LEVO_NA_VPENJANJU;
	"dbDigitalSensors".START_DESNO_NA_VPENJANJU.Input                   := "dbDI".START_DESNO_NA_VPENJANJU;
	"dbDigitalSensors".PRISOTNOST_ZRAKA_NA_NAPRAVI.Input                := "dbDI".PRISOTNOST_ZRAKA_NA_NAPRAVI;
	"dbDigitalSensors".BIMETAL_VIJACENJA_NOGIC_IZKLJUCIL.Input          := "dbDI".BIMETAL_VIJACENJA_NOGIC_IZKLJUCIL;
	"dbDigitalSensors".VIBRATOR_NOGIC_READY.Input                       := "dbDI".VIBRATOR_NOGIC_READY;
	"dbDigitalSensors".BIMETAL_VIJACENJA_NOGIC_IZKLJUCIL.Input          := "dbDI".BIMETAL_VIJACENJA_NOGIC_IZKLJUCIL;
	"dbDigitalSensors".FR_MOTORJA1_ZADAJ_DESNO_READY.Input              := "dbDI".FR_MOTORJA1_ZADAJ_DESNO_READY;
	"dbDigitalSensors".FR_MOTORJA2_SPREDAJ_DESNO_READY.Input            := "dbDI".FR_MOTORJA2_SPREDAJ_DESNO_READY;
	"dbDigitalSensors".FR_MOTORJA1_ZADAJ_LEVO_READY.Input               := "dbDI".FR_MOTORJA1_ZADAJ_LEVO_READY;
	"dbDigitalSensors".FR_MOTORJA2_SPREDAJ_LEVO_READY.Input             := "dbDI".FR_MOTORJA2_SPREDAJ_LEVO_READY;
	"dbDigitalSensors".Spare20_7.Input                                  := "dbDI".Spare20_7;
	"dbDigitalSensors".FOTOCELICA_TRANSPORTA_NOGIC.Input                := "dbDI".FOTOCELICA_TRANSPORTA_NOGIC;
	"dbDigitalSensors".FOTOCELICA_VSTOP_DRCA_NOGIC.Input                := "dbDI".FOTOCELICA_VSTOP_DRCA_NOGIC;
	"dbDigitalSensors".FOTOCELICA_PRED_MESTOM_LOCEVANJA.Input           := "dbDI".FOTOCELICA_PRED_MESTOM_LOCEVANJA;
	"dbDigitalSensors".FOTOCELICA_VSTOP_DRCA_LEVO.Input                 := "dbDI".FOTOCELICA_VSTOP_DRCA_LEVO;
	"dbDigitalSensors".FOTOCELICA_VSTOP_DRCA_DESNO.Input                := "dbDI".FOTOCELICA_VSTOP_DRCA_DESNO;
	"dbDigitalSensors".FOTOCELICA_LOC_IZH_DRCA_LEVO.Input               := "dbDI".FOTOCELICA_LOC_IZH_DRCA_LEVO;
	"dbDigitalSensors".FOTOCELICA_LOC_IZH_DRCA_DESNO.Input              := "dbDI".FOTOCELICA_LOC_IZH_DRCA_DESNO;
	"dbDigitalSensors".NOGICE_V_VIBRATORJU.Input                        := "dbDI".NOGICE_V_VIBRATORJU;
	"dbDigitalSensors".ROTACIJSKI_CIL_DESNO.Input                       := "dbDI".ROTACIJSKI_CIL_DESNO;
	"dbDigitalSensors".ROTACIJSKI_CIL_SREDINA.Input                     := "dbDI".ROTACIJSKI_CIL_SREDINA;
	"dbDigitalSensors".ROTACIJSKI_CIL_LEVO.Input                        := "dbDI".ROTACIJSKI_CIL_LEVO;
	"dbDigitalSensors".LOC_DRCA_DESNO_NAPREJ.Input                      := "dbDI".LOC_DRCA_DESNO_NAPREJ;
	"dbDigitalSensors".LOC_DRCA_DESNO_NAZAJ.Input                       := "dbDI".LOC_DRCA_DESNO_NAZAJ;
	"dbDigitalSensors".LOC_DRCA_LEVO_NAZAJ.Input                        := "dbDI".LOC_DRCA_LEVO_NAZAJ;
	"dbDigitalSensors".LOC_DRCA_LEVO_NAPREJ.Input                       := "dbDI".LOC_DRCA_LEVO_NAPREJ;
	"dbDigitalSensors".Spare22_7.Input                                  := "dbDI".Spare22_7;
	"dbDigitalSensors".FOTOCELICA_LOC_TRAK_DESNO1.Input                := "dbDI".FOTOCELICA_LOC_TRAK_DESNO1;
	"dbDigitalSensors".FOTOCELICA_LOC_TRAK_DESNO2.Input                := "dbDI".FOTOCELICA_LOC_TRAK_DESNO2;
	"dbDigitalSensors".FOTOCELICA_VIJACENJE_DESNOZADAJ.Input            := "dbDI".FOTOCELICA_VIJACENJE_DESNOZADAJ;
	"dbDigitalSensors".FOTOCELICA_VIJACENJE_DESNOSPREDAJ.Input          := "dbDI".FOTOCELICA_VIJACENJE_DESNOSPREDAJ;
	"dbDigitalSensors".VIJACENJE_DESNO_1_NAZAJ.Input                    := "dbDI".VIJACENJE_DESNO_1_NAZAJ;
	"dbDigitalSensors".VIJACENJE_DESNO_1_NAPREJ.Input                   := "dbDI".VIJACENJE_DESNO_1_NAPREJ;
	"dbDigitalSensors".MESTO_VIJAC_STOP_DESNO_ZAD_NAZAJ.Input            := "dbDI".MESTO_VIJAC_STOP_DESNO_ZAD_NAZAJ;
	"dbDigitalSensors".MESTO_VIJAC_STOP_DESNO_ZAD_NAPREJ.Input           := "dbDI".MESTO_VIJAC_STOP_DESNO_ZAD_NAPREJ;
	"dbDigitalSensors".MESTO_VIJACENJE_DESNO_ZAD_DVIG_DOL.Input         := "dbDI".MESTO_VIJACENJE_DESNO_ZAD_DVIG_DOL;
	"dbDigitalSensors".MESTO_VIJACENJE_DESNO_ZAD_CENT_NARAZEN.Input     := "dbDI".MESTO_VIJACENJE_DESNO_ZAD_CENT_NARAZEN;
	"dbDigitalSensors".MESTO_VIJACENJE_DESNO_ZAD_CENT_SKUPAJ.Input      := "dbDI".MESTO_VIJACENJE_DESNO_ZAD_CENT_SKUPAJ;
	"dbDigitalSensors".Spare24_3.Input          := "dbDI".Spare24_3;
	"dbDigitalSensors".Spare24_4.Input         := "dbDI".Spare24_4;
	"dbDigitalSensors".MESTO_VIJACENJE_DESNO_SPRED_DVIG_DOL.Input       := "dbDI".MESTO_VIJACENJE_DESNO_SPRED_DVIG_DOL;
	"dbDigitalSensors".MESTO_VIJACENJE_DESNO_SPRED_CENT_NARAZEN.Input   := "dbDI".MESTO_VIJACENJE_DESNO_SPRED_CENT_NARAZEN;
	"dbDigitalSensors".MESTO_VIJACENJE_DESNO_SPRED_CENT_SKUPAJ.Input    := "dbDI".MESTO_VIJACENJE_DESNO_SPRED_CENT_SKUPAJ;
	"dbDigitalSensors".KONCNA_POZICIJA_VIJACENJA_DES_NAZAJ.Input        := "dbDI".KONCNA_POZICIJA_VIJACENJA_DES_NAZAJ;
	"dbDigitalSensors".KONCNA_POZICIJA_VIJACENJA_DES_NAPREJ.Input       := "dbDI".KONCNA_POZICIJA_VIJACENJA_DES_NAPREJ;
	"dbDigitalSensors".Spare25_2.Input                                  := "dbDI".Spare25_2;
	"dbDigitalSensors".Spare25_3.Input                                  := "dbDI".Spare25_3;
	"dbDigitalSensors".KONCNA_POZICIJA_VIJACENJA_LEVO_NAZAJ.Input       := "dbDI".KONCNA_POZICIJA_VIJACENJA_LEVO_NAZAJ;
	"dbDigitalSensors".KONCNA_POZICIJA_VIJACENJA_LEVO_NAPREJ.Input      := "dbDI".KONCNA_POZICIJA_VIJACENJA_LEVO_NAPREJ;
	"dbDigitalSensors".Spare25_6.Input                                  := "dbDI".Spare25_6;
	"dbDigitalSensors".Spare25_7.Input                                  := "dbDI".Spare25_7;
	"dbDigitalSensors".FOTOCELICA_LOC_TRAK_LEVO1.Input                := "dbDI".FOTOCELICA_LOC_TRAK_LEVO1;
	"dbDigitalSensors".FOTOCELICA_LOC_TRAK_LEVO2.Input                := "dbDI".FOTOCELICA_LOC_TRAK_LEVO2;
	"dbDigitalSensors".FOTOCELICA_VIJACENJE_LEVO_ZADAJ.Input            := "dbDI".FOTOCELICA_VIJACENJE_LEVO_ZADAJ;
	"dbDigitalSensors".FOTOCELICA_VIJACENJE_LEVO_SPREDAJ.Input          := "dbDI".FOTOCELICA_VIJACENJE_LEVO_SPREDAJ;
	"dbDigitalSensors".VIJACENJE_LEVO_1_NAZAJ.Input                     := "dbDI".VIJACENJE_LEVO_1_NAZAJ;
	"dbDigitalSensors".VIJACENJE_LEVO_1_NAPREJ.Input                    := "dbDI".VIJACENJE_LEVO_1_NAPREJ;
	"dbDigitalSensors".MESTO_VIJAC_STOP_LEVO_ZAD_NAZAJ.Input             := "dbDI".MESTO_VIJAC_STOP_LEVO_ZAD_NAZAJ;
	"dbDigitalSensors".MESTO_VIJAC_STOP_LEVO_ZAD_NAPREJ.Input            := "dbDI".MESTO_VIJAC_STOP_LEVO_ZAD_NAPREJ;
	"dbDigitalSensors".MESTO_VIJACENJE_LEVO_ZAD_DVIG_DOL.Input          := "dbDI".MESTO_VIJACENJE_LEVO_ZAD_DVIG_DOL;
	"dbDigitalSensors".MESTO_VIJACENJE_LEVO_ZAD_CENT_NARAZEN.Input      := "dbDI".MESTO_VIJACENJE_LEVO_ZAD_CENT_NARAZEN;
	"dbDigitalSensors".MESTO_VIJACENJE_LEVO_ZAD_CENT_SKUPAJ.Input       := "dbDI".MESTO_VIJACENJE_LEVO_ZAD_CENT_SKUPAJ;
	"dbDigitalSensors".Spare27_3.Input           := "dbDI".Spare27_3;
	"dbDigitalSensors".Spare27_4.Input          := "dbDI".Spare27_4;
	"dbDigitalSensors".MESTO_VIJACENJE_LEVO_SPRED_DVIG_DOL.Input        := "dbDI".MESTO_VIJACENJE_LEVO_SPRED_DVIG_DOL;
	"dbDigitalSensors".MESTO_VIJACENJE_LEVO_SPRED_CENT_NARAZEN.Input    := "dbDI".MESTO_VIJACENJE_LEVO_SPRED_CENT_NARAZEN;
	"dbDigitalSensors".MESTO_VIJACENJE_LEVO_SPRED_CENT_SKUPAJ.Input     := "dbDI".MESTO_VIJACENJE_LEVO_SPRED_CENT_SKUPAJ;
	"dbDigitalSensors".INDUKTIVEC_PRAVILNA_VLOZITEV_DNA_1.Input         := "dbDI".INDUKTIVEC_PRAVILNA_VLOZITEV_DNA_1;
	"dbDigitalSensors".INDUKTIVEC_PRAVILNA_VLOZITEV_DNA_2.Input         := "dbDI".INDUKTIVEC_PRAVILNA_VLOZITEV_DNA_2;
	"dbDigitalSensors".VPENJANJE_DNA_LEVO_ZADAJ_GOR.Input               := "dbDI".VPENJANJE_DNA_LEVO_ZADAJ_GOR;
	"dbDigitalSensors".VPENJANJE_DNA_LEVO_ZADAJ_DOL.Input               := "dbDI".VPENJANJE_DNA_LEVO_ZADAJ_DOL;
	"dbDigitalSensors".VPENJANJE_DNA_LEVO_SPREDAJ_GOR.Input             := "dbDI".VPENJANJE_DNA_LEVO_SPREDAJ_GOR;
	"dbDigitalSensors".VPENJANJE_DNA_LEVO_SPREDAJ_DOL.Input             := "dbDI".VPENJANJE_DNA_LEVO_SPREDAJ_DOL;
	"dbDigitalSensors".VPENJANJE_DNA_DESNO_ZADAJ_GOR.Input              := "dbDI".VPENJANJE_DNA_DESNO_ZADAJ_GOR;
	"dbDigitalSensors".VPENJANJE_DNA_DESNO_ZADAJ_DOL.Input              := "dbDI".VPENJANJE_DNA_DESNO_ZADAJ_DOL;
	"dbDigitalSensors".VPENJANJE_DNA_DESNO_SPREDAJ_GOR.Input            := "dbDI".VPENJANJE_DNA_DESNO_SPREDAJ_GOR;
	"dbDigitalSensors".VPENJANJE_DNA_DESNO_SPREDAJ_DOL.Input            := "dbDI".VPENJANJE_DNA_DESNO_SPREDAJ_DOL;
	
	//----------------------------------------------------------------------
	//  fc call
	//  "cmDigitalSensor"(SimulateEn:=#Simulate,
	"cmDigitalSensor"(Sensor := "dbDigitalSensors".ZAUSTAVITEV_V_SILI_NI_AKTIVIRANA);
	"cmDigitalSensor"(Sensor := "dbDigitalSensors".FOTO_ZAVESA_KANAL_1);
	"cmDigitalSensor"(Sensor := "dbDigitalSensors".FOTO_ZAVESA_KANAL_2);
	"cmDigitalSensor"(Sensor := "dbDigitalSensors".START_LEVO_NA_VPENJANJU);
	"cmDigitalSensor"(Sensor := "dbDigitalSensors".START_DESNO_NA_VPENJANJU);
	"cmDigitalSensor"(Sensor := "dbDigitalSensors".PRISOTNOST_ZRAKA_NA_NAPRAVI);
	"cmDigitalSensor"(Sensor := "dbDigitalSensors".BIMETAL_VIJACENJA_NOGIC_IZKLJUCIL);
	"cmDigitalSensor"(Sensor:="dbDigitalSensors".VIBRATOR_NOGIC_READY);
	"cmDigitalSensor"(Sensor:="dbDigitalSensors".BIMETAL_VIJACENJA_NOGIC_IZKLJUCIL);
	"cmDigitalSensor"(Sensor:="dbDigitalSensors".FR_MOTORJA1_ZADAJ_DESNO_READY);
	"cmDigitalSensor"(Sensor:="dbDigitalSensors".FR_MOTORJA2_SPREDAJ_DESNO_READY);
	"cmDigitalSensor"(Sensor:="dbDigitalSensors".FR_MOTORJA1_ZADAJ_LEVO_READY);
	"cmDigitalSensor"(Sensor:="dbDigitalSensors".FR_MOTORJA2_SPREDAJ_LEVO_READY);
	"cmDigitalSensor"(Sensor := "dbDigitalSensors".Spare20_7);
	"cmDigitalSensor"(Sensor := "dbDigitalSensors".FOTOCELICA_TRANSPORTA_NOGIC);
	"cmDigitalSensor"(Sensor := "dbDigitalSensors".FOTOCELICA_VSTOP_DRCA_NOGIC);
	"cmDigitalSensor"(Sensor := "dbDigitalSensors".FOTOCELICA_PRED_MESTOM_LOCEVANJA);
	"cmDigitalSensor"(Sensor := "dbDigitalSensors".FOTOCELICA_VSTOP_DRCA_LEVO);
	"cmDigitalSensor"(Sensor := "dbDigitalSensors".FOTOCELICA_VSTOP_DRCA_DESNO);;
	"cmDigitalSensor"(Sensor := "dbDigitalSensors".FOTOCELICA_LOC_IZH_DRCA_LEVO);
	"cmDigitalSensor"(Sensor := "dbDigitalSensors".FOTOCELICA_LOC_IZH_DRCA_DESNO);
	"cmDigitalSensor"(Sensor := "dbDigitalSensors".NOGICE_V_VIBRATORJU);
	"cmDigitalSensor"(Sensor := "dbDigitalSensors".ROTACIJSKI_CIL_DESNO);
	"cmDigitalSensor"(Sensor := "dbDigitalSensors".ROTACIJSKI_CIL_SREDINA);
	"cmDigitalSensor"(Sensor := "dbDigitalSensors".ROTACIJSKI_CIL_LEVO);
	"cmDigitalSensor"(Sensor := "dbDigitalSensors".LOC_DRCA_DESNO_NAPREJ);
	"cmDigitalSensor"(Sensor := "dbDigitalSensors".LOC_DRCA_DESNO_NAZAJ);
	"cmDigitalSensor"(Sensor := "dbDigitalSensors".LOC_DRCA_LEVO_NAZAJ);
	"cmDigitalSensor"(Sensor := "dbDigitalSensors".LOC_DRCA_LEVO_NAPREJ);
	"cmDigitalSensor"(Sensor := "dbDigitalSensors".Spare22_7);;
	"cmDigitalSensor"(Sensor := "dbDigitalSensors".FOTOCELICA_LOC_TRAK_DESNO1);;
	"cmDigitalSensor"(Sensor := "dbDigitalSensors".FOTOCELICA_LOC_TRAK_DESNO2);
	"cmDigitalSensor"(Sensor := "dbDigitalSensors".FOTOCELICA_VIJACENJE_DESNOZADAJ);
	"cmDigitalSensor"(Sensor := "dbDigitalSensors".FOTOCELICA_VIJACENJE_DESNOSPREDAJ);
	"cmDigitalSensor"(Sensor := "dbDigitalSensors".VIJACENJE_DESNO_1_NAZAJ);
	"cmDigitalSensor"(Sensor := "dbDigitalSensors".VIJACENJE_DESNO_1_NAPREJ);
	"cmDigitalSensor"(Sensor := "dbDigitalSensors".MESTO_VIJAC_STOP_DESNO_ZAD_NAZAJ);
	"cmDigitalSensor"(Sensor := "dbDigitalSensors".MESTO_VIJAC_STOP_DESNO_ZAD_NAPREJ);
	"cmDigitalSensor"(Sensor := "dbDigitalSensors".MESTO_VIJACENJE_DESNO_ZAD_DVIG_DOL);
	"cmDigitalSensor"(Sensor := "dbDigitalSensors".MESTO_VIJACENJE_DESNO_ZAD_CENT_NARAZEN);
	"cmDigitalSensor"(Sensor := "dbDigitalSensors".MESTO_VIJACENJE_DESNO_ZAD_CENT_SKUPAJ);
	"cmDigitalSensor"(Sensor := "dbDigitalSensors".Spare24_3);
	"cmDigitalSensor"(Sensor := "dbDigitalSensors".Spare24_4);
	"cmDigitalSensor"(Sensor := "dbDigitalSensors".MESTO_VIJACENJE_DESNO_SPRED_DVIG_DOL);;
	"cmDigitalSensor"(Sensor := "dbDigitalSensors".MESTO_VIJACENJE_DESNO_SPRED_CENT_NARAZEN);
	"cmDigitalSensor"(Sensor := "dbDigitalSensors".MESTO_VIJACENJE_DESNO_SPRED_CENT_SKUPAJ);
	"cmDigitalSensor"(Sensor := "dbDigitalSensors".KONCNA_POZICIJA_VIJACENJA_DES_NAZAJ);
	"cmDigitalSensor"(Sensor := "dbDigitalSensors".KONCNA_POZICIJA_VIJACENJA_DES_NAPREJ);
	"cmDigitalSensor"(Sensor := "dbDigitalSensors".Spare25_2);
	"cmDigitalSensor"(Sensor := "dbDigitalSensors".Spare25_3);
	"cmDigitalSensor"(Sensor := "dbDigitalSensors".KONCNA_POZICIJA_VIJACENJA_LEVO_NAZAJ);
	"cmDigitalSensor"(Sensor := "dbDigitalSensors".KONCNA_POZICIJA_VIJACENJA_LEVO_NAPREJ);
	"cmDigitalSensor"(Sensor := "dbDigitalSensors".Spare25_6);
	"cmDigitalSensor"(Sensor := "dbDigitalSensors".Spare25_7);
	"cmDigitalSensor"(Sensor := "dbDigitalSensors".FOTOCELICA_LOC_TRAK_LEVO1);
	"cmDigitalSensor"(Sensor := "dbDigitalSensors".FOTOCELICA_LOC_TRAK_LEVO2);
	"cmDigitalSensor"(Sensor := "dbDigitalSensors".FOTOCELICA_VIJACENJE_LEVO_ZADAJ);
	"cmDigitalSensor"(Sensor := "dbDigitalSensors".FOTOCELICA_VIJACENJE_LEVO_SPREDAJ);
	"cmDigitalSensor"(Sensor:="dbDigitalSensors".VIJACENJE_LEVO_1_NAZAJ);
	"cmDigitalSensor"(Sensor:="dbDigitalSensors".VIJACENJE_LEVO_1_NAPREJ);
	"cmDigitalSensor"(Sensor := "dbDigitalSensors".MESTO_VIJAC_STOP_LEVO_ZAD_NAZAJ);
	"cmDigitalSensor"(Sensor := "dbDigitalSensors".MESTO_VIJAC_STOP_LEVO_ZAD_NAPREJ);
	"cmDigitalSensor"(Sensor := "dbDigitalSensors".MESTO_VIJACENJE_LEVO_ZAD_DVIG_DOL);
	"cmDigitalSensor"(Sensor := "dbDigitalSensors".MESTO_VIJACENJE_LEVO_ZAD_CENT_NARAZEN);
	"cmDigitalSensor"(Sensor := "dbDigitalSensors".MESTO_VIJACENJE_LEVO_ZAD_CENT_SKUPAJ);
	"cmDigitalSensor"(Sensor := "dbDigitalSensors".Spare27_3);
	"cmDigitalSensor"(Sensor := "dbDigitalSensors".Spare27_4);
	"cmDigitalSensor"(Sensor := "dbDigitalSensors".MESTO_VIJACENJE_LEVO_SPRED_DVIG_DOL);
	"cmDigitalSensor"(Sensor := "dbDigitalSensors".MESTO_VIJACENJE_LEVO_SPRED_CENT_NARAZEN);
	"cmDigitalSensor"(Sensor := "dbDigitalSensors".MESTO_VIJACENJE_LEVO_SPRED_CENT_SKUPAJ);
	"cmDigitalSensor"(Sensor := "dbDigitalSensors".INDUKTIVEC_PRAVILNA_VLOZITEV_DNA_1);
	"cmDigitalSensor"(Sensor := "dbDigitalSensors".INDUKTIVEC_PRAVILNA_VLOZITEV_DNA_2);
	"cmDigitalSensor"(Sensor := "dbDigitalSensors".VPENJANJE_DNA_LEVO_ZADAJ_GOR);
	"cmDigitalSensor"(Sensor := "dbDigitalSensors".VPENJANJE_DNA_LEVO_ZADAJ_DOL);
	"cmDigitalSensor"(Sensor := "dbDigitalSensors".VPENJANJE_DNA_LEVO_SPREDAJ_GOR);
	"cmDigitalSensor"(Sensor := "dbDigitalSensors".VPENJANJE_DNA_LEVO_SPREDAJ_DOL);
	"cmDigitalSensor"(Sensor := "dbDigitalSensors".VPENJANJE_DNA_DESNO_ZADAJ_GOR);
	"cmDigitalSensor"(Sensor := "dbDigitalSensors".VPENJANJE_DNA_DESNO_ZADAJ_DOL);
	"cmDigitalSensor"(Sensor := "dbDigitalSensors".VPENJANJE_DNA_DESNO_SPREDAJ_GOR);
	"cmDigitalSensor"(Sensor := "dbDigitalSensors".VPENJANJE_DNA_DESNO_SPREDAJ_DOL);
	"cmDigitalSensor"(Sensor := "dbDigitalSensors".NOGICE_V_VIBRATORJU);
END_FUNCTION

FUNCTION "cmDigitalSensor" : Void
{ S7_Optimized_Access := 'FALSE' }
VERSION : 0.1
   VAR_IN_OUT 
      Sensor : "udtDigitalSensor";
   END_VAR

   VAR_TEMP 
      tmpTimer : Int;
      tmpTimerDelay : Int;
   END_VAR


BEGIN
	//----------------------------------------------------------------------   
	// init timers
	#tmpTimer := CHAR_TO_INT(BYTE_TO_CHAR(#Sensor.Timer1));
	#tmpTimerDelay := CHAR_TO_INT(BYTE_TO_CHAR(#Sensor.FilterTime));
	
	IF #Sensor.ManOn = 1 OR #Sensor.ManOff = 1 THEN
	    #Sensor.Manual := True;
	    IF #Sensor.ManOn THEN
	        IF NOT #Sensor.Invert THEN
	            #Sensor.Input := True;
	        ELSE
	            #Sensor.Input := False;
	        END_IF;
	    ELSIF #Sensor.ManOff THEN
	        IF NOT #Sensor.Invert THEN
	            #Sensor.Input := False;
	        ELSE
	            #Sensor.Input := True;
	        END_IF;
	    END_IF;
	ELSE
	    #Sensor.Manual := False;
	END_IF;
	
	// reset timer
	IF (NOT #Sensor.Invert AND #Sensor.Input = #Sensor.InputF) OR (#Sensor.Invert AND #Sensor.Input <> #Sensor.InputF) THEN
	    #Sensor.Timer1 := 0;
	END_IF;
	
	// change of DI raw value
	IF (NOT #Sensor.Invert AND #Sensor.Input <> #Sensor.InputF) OR (#Sensor.Invert AND #Sensor.Input = #Sensor.InputF) THEN
	    
	    // filter time
	    IF "100msOSR" AND #tmpTimer < #tmpTimerDelay THEN
	        #tmpTimer := #tmpTimer + 1;
	        #Sensor.Timer1 := CHAR_TO_BYTE(INT_TO_CHAR(#tmpTimer));
	    END_IF;
	    
	    // filter time ends
	    IF #tmpTimer >= #tmpTimerDelay THEN
	        IF #Sensor.Invert THEN
	            #Sensor.InputF := NOT (#Sensor.Input);
	        ELSE
	            #Sensor.InputF := #Sensor.Input;
	        END_IF;
	    END_IF;
	END_IF;
	
	// OSR
	#Sensor.OSR := FALSE;
	IF #Sensor.Input <> #Sensor.OSRHist AND #Sensor.Input THEN
	    #Sensor.OSR := TRUE;
	END_IF;
	#Sensor.OSRHist := #Sensor.Input;
	
	// OSF
	#Sensor.OSF := FALSE;
	IF #Sensor.Input <> #Sensor.OSFHist AND NOT #Sensor.Input THEN
	    #Sensor.OSF := TRUE;
	END_IF;
	#Sensor.OSFHist := #Sensor.Input;
	
END_FUNCTION

FUNCTION "fcHSCEncoder" : Void
{ S7_Optimized_Access := 'TRUE' }
VERSION : 0.1

BEGIN
	// Short summary:
	(*
	  fcHSCEncoders - call encoders funcions
	*)
	// 
	//**********************************************************************
	// Revision control:
	//----------------------------------------------------------------------
	// Use only for revisions of original code
	// V0.01
	// Description of revision
	
	//----------------------------------------------------------------------
	// Comments:
	(*
	  Every change in the code is documented with following:
	  // CCC-yyymmdd: .....
	  yyyy year when change was made
	  mm   month when change was made
	  dd   day when change was made
	  CCC  authors initials
	*)
	
	// NOT IN USE
	(*
	"cmHSC"(HdrAdr:=257,
	        Direction:="dbHSC".ScanLineCounts.Direction,
	        CV:="dbHSC".ScanLineCounts.CV,
	        RV:="dbHSC".ScanLineCounts.RV,
	        Period:="dbHSC".ScanLineCounts.Period,
	        New_dir:="dbHSC".ScanLineCounts.New_dir,
	        New_CV:="dbHSC".ScanLineCounts.New_CV,
	        New_RV:="dbHSC".ScanLineCounts.New_RV,
	        New_period:="dbHSC".ScanLineCounts.New_period,
	        HdrAdr_Counter := "cmHSC_HdrAdr_Counter1",
	        Busy=>"dbHSC".ScanLineCounts.Busy,
	        Status=>"dbHSC".ScanLineCounts.Status,
	        CounterValue=>"dbHSC".ScanLineCounts.CounterValue);
	"dbHSC".ScanLineCounts.CounterValueReal := "dbHSC".ScanLineCounts.CounterValue;
	"dbHSC".ScanLineCounts.EguValue := "dbHSC".ScanLineCounts.CounterValueReal / "dbHSC".ScanLineCounts.EguFactor;
	*)
END_FUNCTION

FUNCTION "cmHSC" : Void
{ S7_Optimized_Access := 'FALSE' }
VERSION : 0.1
   VAR_INPUT 
      HdrAdr : HW_HSC;
      Direction : Bool;
      CV : Bool;
      RV : Bool;
      Period : Bool;
      New_dir : Int;
      New_CV : DInt;
      New_RV : DInt;
      New_period : Int;
      HdrAdr_Counter : DWord;
   END_VAR

   VAR_OUTPUT 
      Busy : Bool;
      Status : Word;
      CounterValue : DWord;
   END_VAR

   VAR_TEMP 
      i : Int;
   END_VAR


BEGIN
	"CTRL_HSC_0_DB"(HSC:=#HdrAdr,
	                DIR:=#Direction,
	                CV:=#CV,
	                RV:=#RV,
	                PERIOD:=#Period,
	                NEW_DIR:=#New_dir,
	                NEW_CV:=#New_CV,
	                NEW_RV:=#New_RV,
	                NEW_PERIOD:=#New_period,
	                BUSY=>#Busy,
	                STATUS=>#Status);
	#CounterValue := #HdrAdr_Counter;
END_FUNCTION

FUNCTION "fcSystemAlarms" : Void
{ S7_Optimized_Access := 'FALSE' }
VERSION : 0.1
   VAR_TEMP 
      z : Int;
      k : Int;
      i : Int;
      j : Int;
      m : Int;
   END_VAR


BEGIN
	// Short summary:
	(*
	  Alarms that stop the whole system
	*)
	// 
	//**********************************************************************
	// Revision control:
	//----------------------------------------------------------------------
	// Use only for revisions of original code
	// V0.01
	// Description of revision
	
	//----------------------------------------------------------------------
	// Comments:
	(*
	  Every change in the code is documented with following:
	  // CCC-yyymmdd: .....
	  yyyy year when change was made
	  mm   month when change was made
	  dd   day when change was made
	  CCC  authors initials
	*)
	//**********************************************************************
	IF "AlarmAck" THEN
	    FOR #z := 1 TO 1024 BY 1 DO
	        "dbSystemAlarms".SysAlm[#z] := False;
	    END_FOR;
	END_IF;
	
	// System Alarm  - Emergency stop,...
	"dbSystemAlarms".SysAlm[01] := NOT "dbDigitalSensors".ZAUSTAVITEV_V_SILI_NI_AKTIVIRANA.InputF;
	"dbSystemAlarms".SysAlm[02] := NOT "dbDigitalSensors".PRISOTNOST_ZRAKA_NA_NAPRAVI.InputF;
	
	"dbSystemAlarms".SysAlm[03] := NOT "dbDigitalSensors".FOTO_ZAVESA_KANAL_1.InputF;
	"dbSystemAlarms".SysAlm[04] := NOT "dbDigitalSensors".FOTO_ZAVESA_KANAL_2.InputF;
	"dbSystemAlarms".SysAlm[05] := NOT "dbDigitalSensors".FOTO_ZAVESA_KANAL_1.InputF OR NOT "dbDigitalSensors".FOTO_ZAVESA_KANAL_2.InputF; // Used on HMI
END_FUNCTION

FUNCTION "fcResetAvto" : Void
{ S7_Optimized_Access := 'FALSE' }
VERSION : 0.1

BEGIN
	// Short summary:
	(*
	  Reset of control elements performed every cycle
	*)
	// 
	//**********************************************************************
	// Revision control:
	//----------------------------------------------------------------------
	// Use only for revisions of original code
	// V0.01
	// Description of revision
	
	//----------------------------------------------------------------------
	// Comments:
	(*
	  Every change in the code is documented with following:
	  // CCC-yyymmdd: .....
	  yyyy year when change was made
	  mm   month when change was made
	  dd   day when change was made
	  CCC  authors initials
	*)
	//**********************************************************************
	
	//----------------------------------------------------------------------
	//  DigitalValves
	"dbDigitalValves".Y17_RotCilipozDesno.AutoON       := False;
	"dbDigitalValves".Y18_RotCilipozLevo.AutoON        := False;
	"dbDigitalValves".Y2_VijaDesZad_Dvig.AutoON       := False;
	"dbDigitalValves".Y3_VijaDesSpr_Dvig.AutoON       := False;
	"dbDigitalValves".Y4_VijaLevZad_Dvig.AutoON      := False;
	"dbDigitalValves".Y5_VijaLevSpr_Dvig.AutoON      := False;
	"dbDigitalValves".Y6_DrcaLocev_Des.AutoON         := False;
	"dbDigitalValves".Y7_DrcaLocev_Lev.AutoON         := False;
	"dbDigitalValves".Y8_VijaLocev_Des.AutoON         := False;
	"dbDigitalValves".Y9_VijaStop_DesZad.AutoON       := False;
	"dbDigitalValves".Y10_Centri_DesZad.AutoON         := False;
	"dbDigitalValves".Y11_Centri_DesSpr.AutoON        := False;
	"dbDigitalValves".Y12_VijaLocev_Lev.AutoON        := False;
	"dbDigitalValves".Y13_VijaStop_LevZad.AutoON      := False;
	"dbDigitalValves".Y14_Centri_LevZad.AutoON        := False;
	"dbDigitalValves".Y15_Centri_LevSpr.AutoON        := False;
	"dbDigitalValves".Y16_VpenjanjeDna.AutoON         := False;
	"dbDigitalValves".SEMAFOR_ZELENA.AutoON           := False;
	"dbDigitalValves".SEMAFOR_RUMENA.AutoON           := False;
	"dbDigitalValves".SEMAFOR_RDECA.AutoON            := False;
	//----------------------------------------------------------------------
	
	//----------------------------------------------------------------------
	//  Motors
	"dbMotors".VKLOP_M_TRACNEGA_TRANS_NOGIC.AutoON      := False;
	"dbMotors".M1_ZADAJ_DESNO.AutoON                    := False;
	"dbMotors".M2_SPREDAJ_DESNO.AutoON                  := False;
	"dbMotors".M1_ZADAJ_LEVO.AutoON                     := False;
	"dbMotors".M2_SPREDAJ_LEVO.AutoON                   := False;
	"dbMotors".VKLOP_VIBRATORJA.AutoON                  := False;
	"dbMotors".VKLOP_M_TRAKA_VIJACNIKA.AutoON           := False;
END_FUNCTION

FUNCTION "fcOPAlarming" : Void
{ S7_Optimized_Access := 'FALSE' }
VERSION : 0.1
   VAR_TEMP 
      i : Int;
      j : Int;
      WordTmp1 : Word;
      WordTmp2 : Word;
   END_VAR


BEGIN
	//-------------------------------------------------------------------------------------------------
	// reset alarms
	IF "AlarmAck" THEN
	(*
	  "dbProfinetAlrm".ULS_HMIAlarm_WDT := 0;
	  "dbProfinetAlrm".LS_HMIAlarm_WDT := 0;
	  "dbProfinetAlrm".LS_HMIAlarm_Bit := False;
	  "dbProfinetAlrm".ULS_HMIAlarm_Bit := False;
	  "dbProfinetAlrm".ProfinetAlarm := False;
	  *)
	    FOR #i := 0 TO 63 BY 1 DO
	      "dbOPAlarms".Alarm[#i] := false;
	  END_FOR;
	END_IF;
	//-------------------------------------------------------------------------------------------------
	
	// #Y8_VijaLocev_Des
	"dbOPAlarms".Alarm[0] := "dbAlarms".PLI[1, 1];
	
	// #V5_VijaStop_DesZad
	"dbOPAlarms".Alarm[1] := "dbAlarms".PLI[1, 2];
	
	// #V6_VijaDesZad_Dvig
	"dbOPAlarms".Alarm[2] := "dbAlarms".PLI[1, 3];
	
	// #V7_Centri_DesZad
	"dbOPAlarms".Alarm[3] := "dbAlarms".PLI[1, 4];
	
	// #V9_VijaDesSpr_Dvig
	"dbOPAlarms".Alarm[4] := "dbAlarms".PLI[1, 5];
	
	// #V10_Centri_DesSpr
	"dbOPAlarms".Alarm[5] := "dbAlarms".PLI[1, 6];
	
	// #V11_VijaLocev_Lev
	"dbOPAlarms".Alarm[6] := "dbAlarms".PLI[1, 7];
	
	// #V12_VijaStop_LevZad
	"dbOPAlarms".Alarm[7] := "dbAlarms".PLI[1, 8];
	
	// #V13_VijaLevZad_Dvig
	"dbOPAlarms".Alarm[8] := "dbAlarms".PLI[1, 9];
	
	// #V14_Centri_LevZad
	"dbOPAlarms".Alarm[9] := "dbAlarms".PLI[1, 10];
	
	// #V16_VijaLevSpr_Dvig
	"dbOPAlarms".Alarm[10] := "dbAlarms".PLI[1, 11];
	
	// #V17_Centri_LevSpr
	"dbOPAlarms".Alarm[11] := "dbAlarms".PLI[1, 12];
	
	// #V18_VpenjanjeDna
	"dbOPAlarms".Alarm[12] := "dbAlarms".PLI[1, 13];
	
	// #M1_ZADAJ_LEVO
	"dbOPAlarms".Alarm[13] := "dbAlarms".PLI[1, 14];
	
	// #M2_SPREDAJ_LEVO
	"dbOPAlarms".Alarm[14] := "dbAlarms".PLI[1, 15];
	
	// #M1_ZADAJ_DESNO
	"dbOPAlarms".Alarm[15] := "dbAlarms".PLI[1, 16];
	
	// #M2_SPREDAJ_DESNO
	"dbOPAlarms".Alarm[16] := "dbAlarms".PLI[1, 17];
	
	// #VKLOP_M_TRAKA_VIJACNIKA
	"dbOPAlarms".Alarm[17] := "dbAlarms".PLI[1, 18];
	
	// Začetne pozicije vijačnega dela niso dosežene
	"dbOPAlarms".Alarm[28] := "dbAlarms".PLI[1, 19];
	
	// Manjka ena od nogic na pozicijah za vijačenje-ročno odstrani nogice
	"dbOPAlarms".Alarm[31] := "dbAlarms".PLI[1, 20];
	
	// Dovoljeni čas vijačenja nogice levo-spredaj potekel
	"dbOPAlarms".Alarm[32] := "dbAlarms".PLI[1, 21];
	
	// Dovoljeni čas vijačenja nogice levo-zadaj potekel
	"dbOPAlarms".Alarm[33] := "dbAlarms".PLI[1, 22];
	
	// Dovoljeni čas vijačenja nogice desno-spredaj potekel
	"dbOPAlarms".Alarm[34] := "dbAlarms".PLI[1, 23];
	
	// Dovoljeni čas vijačenja nogice desno-zadaj potekel
	"dbOPAlarms".Alarm[35] := "dbAlarms".PLI[1, 24];
	
	// #V1_RotCilipozLevo
	"dbOPAlarms".Alarm[18] := "dbAlarms".PLI[2, 1];
	
	// #V1_RotCilipozDesno
	"dbOPAlarms".Alarm[19] := "dbAlarms".PLI[2, 2];
	
	// #V3_DrcaLocev_Lev
	"dbOPAlarms".Alarm[20] := "dbAlarms".PLI[2, 3];
	
	// #V2_DrcaLocev_Des
	"dbOPAlarms".Alarm[21] := "dbAlarms".PLI[2, 4];
	
	// Začetna pozicija rotacijskega cilindra ni dosežena
	"dbOPAlarms".Alarm[29] := "dbAlarms".PLI[2, 5];
	
	// ZAUSTAVITEV_V_SILI_NI_AKTIVIRANA
	"dbOPAlarms".Alarm[22] := "dbAlarms".PLI[3, 1];
	
	// PRISOTNOST_ZRAKA_NA_NAPRAVI
	"dbOPAlarms".Alarm[23] := "dbAlarms".PLI[3, 2];
	
	// FOTO_ZAVESA_KANAL_1
	"dbOPAlarms".Alarm[24] := "dbAlarms".PLI[3, 3];
	
	// FOTO_ZAVESA_KANAL_2
	"dbOPAlarms".Alarm[25] := "dbAlarms".PLI[3, 4];
	
	// #VKLOP_M_TRACNEGA_TRANS_NOGIC
	"dbOPAlarms".Alarm[26] := "dbAlarms".PLI[3, 5];
	
	// #VKLOP_VIBRATORJA
	"dbOPAlarms".Alarm[27] := "dbAlarms".PLI[3, 6];
	
	// Prisoten eden od alarmov
	"dbOPAlarms".Alarm[30] := "dbAlarms".PLI[3, 7];
	
	// Opozorilo - dodaj nogice v vstopni zalogovnik
	"dbOPAlarms".Alarm[36] := "dbAlarms".PLI[3, 8];
	
	// shift words for OP
	"dbOPAlarms".OPAlarmWord[00] := INT_TO_WORD(BYTE_TO_INT(%DB112.DBB1) * 256 + BYTE_TO_INT(%DB112.DBB0));
	"dbOPAlarms".OPAlarmWord[01] := INT_TO_WORD(BYTE_TO_INT(%DB112.DBB3) * 256 + BYTE_TO_INT(%DB112.DBB2));
	"dbOPAlarms".OPAlarmWord[02] := INT_TO_WORD(BYTE_TO_INT(%DB112.DBB5) * 256 + BYTE_TO_INT(%DB112.DBB4));
	"dbOPAlarms".OPAlarmWord[03] := INT_TO_WORD(BYTE_TO_INT(%DB112.DBB7) * 256 + BYTE_TO_INT(%DB112.DBB6));
	
END_FUNCTION

FUNCTION "fcUnitInterlocks" : Void
{ S7_Optimized_Access := 'FALSE' }
VERSION : 0.1
   VAR_TEMP 
      i : Int;
      GenIntl_1 : Bool;
      GenIntl_2 : Bool;
      GenIntl_3 : Bool;
      GenIntl_4 : Bool;
      GenIntl_5 : Bool;
      GenIntl_6 : Bool;
      GenIntl_7 : Bool;
      GenIntl_8 : Bool;
   END_VAR


BEGIN
	// Short summary:
	(*
	  Unit interlocks
	*)
	// 
	//**********************************************************************
	// Revision control:
	//----------------------------------------------------------------------
	// Use only for revisions of original code
	// V0.01
	// Description of revision
	
	//----------------------------------------------------------------------
	// Comments:
	(*
	  Every change in the code is documented with following:
	  // CCC-yyymmdd: .....
	  yyyy year when change was made
	  mm   month when change was made
	  dd   day when change was made
	  CCC  authors initials
	*)
	//**********************************************************************
	
	//----------------------------------------------------------------------
	//  General Interlock - All Units
	//  System Alarm - Emergency STOP 
	#GenIntl_1       :=     "dbSystemAlarms".SysAlm[1] OR "dbSystemAlarms".SysAlm[2] OR False; // E_STOP + AirSupply
	#GenIntl_2       :=     "dbSystemAlarms".SysAlm[3] OR "dbSystemAlarms".SysAlm[4] OR False; // Safety light curtain
	
	//----------------------------------------------------------------------
	//  DigitalValves
	"dbDigitalValves".Y2_VijaDesZad_Dvig.Interlock      := #GenIntl_1 OR NOT "dbDigitalSensors".MESTO_VIJAC_STOP_DESNO_ZAD_NAPREJ.InputF;
	IF "dbDigitalValves".Y2_VijaDesZad_Dvig.Interlock THEN
	  "dbDigitalValves".Y2_VijaDesZad_Dvig.ManON := False;
	END_IF;
	"dbDigitalValves".Y3_VijaDesSpr_Dvig.Interlock      := #GenIntl_1;
	"dbDigitalValves".Y4_VijaLevZad_Dvig.Interlock      := #GenIntl_1 OR NOT "dbDigitalSensors".MESTO_VIJAC_STOP_LEVO_ZAD_NAPREJ.InputF;
	IF "dbDigitalValves".Y4_VijaLevZad_Dvig.Interlock THEN
	  "dbDigitalValves".Y4_VijaLevZad_Dvig.ManON := False;
	END_IF;
	"dbDigitalValves".Y5_VijaLevSpr_Dvig.Interlock      := #GenIntl_1;
	IF (#GenIntl_1 OR False) THEN
	  "dbPDO".Y2_VijaDesZad_Spust      := FALSE;
	END_IF;
	IF (#GenIntl_1 OR False) THEN
	  "dbPDO".Y3_VijaDesSpr_Spust      := False;
	END_IF;
	IF (#GenIntl_1 OR False) THEN
	  "dbPDO".Y4_VijaLevZad_Spust     := False;
	END_IF;
	IF (#GenIntl_1 OR False) THEN
	  "dbPDO".Y5_VijaLevSpr_Spust     := False;
	END_IF;
	
	"dbDigitalValves".Y6_DrcaLocev_Des.Interlock         := #GenIntl_1;
	"dbDigitalValves".Y7_DrcaLocev_Lev.Interlock         := #GenIntl_1;
	"dbDigitalValves".Y8_VijaLocev_Des.Interlock         := #GenIntl_1;
	
	"dbDigitalValves".Y9_VijaStop_DesZad.Interlock       := #GenIntl_1;
	IF NOT "dbDigitalSensors".MESTO_VIJACENJE_DESNO_ZAD_DVIG_DOL.InputF THEN
	  "dbDigitalValves".Y9_VijaStop_DesZad.Interlock  := True; // prevent to move back, if motor in UP and interlock present
	END_IF;
	
	"dbDigitalValves".Y10_Centri_DesZad.Interlock        := #GenIntl_1;
	"dbDigitalValves".Y11_Centri_DesSpr.Interlock        := #GenIntl_1;
	"dbDigitalValves".Y12_VijaLocev_Lev.Interlock        := #GenIntl_1;
	
	"dbDigitalValves".Y13_VijaStop_LevZad.Interlock      := #GenIntl_1;
	IF NOT "dbDigitalSensors".MESTO_VIJACENJE_LEVO_ZAD_DVIG_DOL.InputF THEN
	  "dbDigitalValves".Y13_VijaStop_LevZad.Interlock  := True; // prevent to move back, if motor in UP and interlock present
	END_IF;
	"dbDigitalValves".Y14_Centri_LevZad.Interlock        := #GenIntl_1;
	"dbDigitalValves".Y15_Centri_LevSpr.Interlock        := #GenIntl_1;
	"dbDigitalValves".Y16_VpenjanjeDna.Interlock         := #GenIntl_1;
	"dbDigitalValves".Y17_RotCilipozDesno.Interlock      := #GenIntl_1 OR ("dbDigitalValves".Y18_RotCilipozLevo.XS)  OR False; // Interlock opposite valve
	IF "dbDigitalSensors".ROTACIJSKI_CIL_DESNO.InputF AND "dbDigitalValves".Y18_RotCilipozLevo.ManON THEN
	  "dbDigitalValves".Y18_RotCilipozLevo.ManON := False; // prenvent move to directlly move from DESNO >>> LEVO. First HMI user needs to press SREDINA
	END_IF;
	
	"dbDigitalValves".Y18_RotCilipozLevo.Interlock       := #GenIntl_1 OR ("dbDigitalValves".Y17_RotCilipozDesno.XS) OR False; // Interlock opposite valve
	IF "dbDigitalSensors".ROTACIJSKI_CIL_LEVO.InputF AND "dbDigitalValves".Y17_RotCilipozDesno.ManON THEN
	  "dbDigitalValves".Y17_RotCilipozDesno.ManON := False; // prenvent move to directlly move from DESNO >>> LEVO. First HMI user needs to press SREDINA
	END_IF;
	
	"dbDigitalValves".SEMAFOR_ZELENA.Interlock           := False;
	"dbDigitalValves".SEMAFOR_RUMENA.Interlock           := False;
	"dbDigitalValves".SEMAFOR_RDECA.Interlock            := False;
	//----------------------------------------------------------------------
	//  Motors
	"dbMotors".VKLOP_M_TRACNEGA_TRANS_NOGIC.Interlock      := #GenIntl_1 OR False;
	"dbMotors".M1_ZADAJ_DESNO.Interlock                    := #GenIntl_1 OR #GenIntl_2;
	"dbMotors".M2_SPREDAJ_DESNO.Interlock                  := #GenIntl_1 OR #GenIntl_2;
	"dbMotors".M1_ZADAJ_LEVO.Interlock                     := #GenIntl_1 OR #GenIntl_2;
	"dbMotors".M2_SPREDAJ_LEVO.Interlock                   := #GenIntl_1 OR #GenIntl_2;
	"dbMotors".VKLOP_VIBRATORJA.Interlock                  := #GenIntl_1 OR False;
	"dbMotors".VKLOP_M_TRAKA_VIJACNIKA.Interlock           := #GenIntl_1; // OR #GenIntl_2 TRAK se ne ustavi če zavesa ni OK
END_FUNCTION

FUNCTION "TIMER_ON_DELAY" : Void
{ S7_Optimized_Access := 'FALSE' }
VERSION : 0.1
   VAR_TEMP 
      i : Int;
      j : Int;
      MAX_TIMER_NO : Int;
   END_VAR


BEGIN
	#i := 0;
	#MAX_TIMER_NO := 10 * "MaxPLITimersIndex";
	
	WHILE (#i <= #MAX_TIMER_NO) DO
	    
	    // timer reset bit = 1 
	    IF "dbTimers".Num[#i].RS THEN
	        "dbTimers".Num[#i].ACC := 0;                           // ACC value = 0
	        "dbTimers".Num[#i].TT := FALSE;                        // timing bit = 0
	        "dbTimers".Num[#i].DN := FALSE;                        // done bit = 0   
	        "dbTimers".Num[#i].RS := FALSE;
	    END_IF;
	    
	    IF "dbTimers".Num[#i].EE THEN
	        // timer enable bit = 1
	        
	        IF "dbTimers".Num[#i].ACC < "dbTimers".Num[#i].PRE AND NOT "dbTimers".Num[#i].FR THEN
	          IF "100msOSR" = TRUE THEN
	            "dbTimers".Num[#i].ACC := "dbTimers".Num[#i].ACC + 1;
	          END_IF;
	          "dbTimers".Num[#i].TT := TRUE;   // PRE < ACC -> timing bit = 1
	          "dbTimers".Num[#i].DN := FALSE;  // PRE < ACC -> done bit = 0               
	        END_IF;
	        
	        IF "dbTimers".Num[#i].ACC >= "dbTimers".Num[#i].PRE THEN
	            "dbTimers".Num[#i].TT := FALSE;  // PRE = ACC -> timing bit = 0
	            "dbTimers".Num[#i].DN := TRUE;   // PRE = ACC -> done bit = 1               
	        END_IF;
	        
	        //      "dbTimers".Num[i].EE := False;
	    ELSE
	        // timer enable bit = 0
	        "dbTimers".Num[#i].ACC := 0;     // ACC = 0
	        "dbTimers".Num[#i].TT := FALSE;  // timing bit = 0
	        "dbTimers".Num[#i].DN := FALSE;  // done bit = 0
	        
	    END_IF;
	    ;
	    
	    #i := #i + 1;
	    
	END_WHILE;
	
END_FUNCTION

FUNCTION "fcImplementation" : Void
{ S7_Optimized_Access := 'TRUE' }
VERSION : 0.1

BEGIN
	"ph_Helix_1_DB"(Y8_VijaLocev_Des:= "dbDigitalValves".Y8_VijaLocev_Des,
	                Y9_VijaStop_DesZad:= "dbDigitalValves".Y9_VijaStop_DesZad,
	                Y2_VijaDesZad_Dvig:= "dbDigitalValves".Y2_VijaDesZad_Dvig,
	                Y10_Centri_DesZad:= "dbDigitalValves".Y10_Centri_DesZad,
	                Y3_VijaDesSpr_Dvig:= "dbDigitalValves".Y3_VijaDesSpr_Dvig,
	                Y11_Centri_DesSpr:= "dbDigitalValves".Y11_Centri_DesSpr,
	                Y12_VijaLocev_Lev:= "dbDigitalValves".Y12_VijaLocev_Lev,
	                Y13_VijaStop_LevZad:= "dbDigitalValves".Y13_VijaStop_LevZad,
	                Y4_VijaLevZad_Dvig:= "dbDigitalValves".Y4_VijaLevZad_Dvig,
	                Y14_Centri_LevZad:= "dbDigitalValves".Y14_Centri_LevZad,
	                Y5_VijaLevSpr_Dvig:= "dbDigitalValves".Y5_VijaLevSpr_Dvig,
	                Y15_Centri_LevSpr:= "dbDigitalValves".Y15_Centri_LevSpr,
	                Y16_VpenjanjeDna:= "dbDigitalValves".Y16_VpenjanjeDna,
	                M1_ZADAJ_LEVO:= "dbMotors".M1_ZADAJ_LEVO,
	                M2_SPREDAJ_LEVO:= "dbMotors".M2_SPREDAJ_LEVO,
	                M1_ZADAJ_DESNO:= "dbMotors".M1_ZADAJ_DESNO,
	                M2_SPREDAJ_DESNO:= "dbMotors".M2_SPREDAJ_DESNO,
	                VKLOP_M_TRAKA_VIJACNIKA:="dbMotors".VKLOP_M_TRAKA_VIJACNIKA);
	
	"ph_LegsShifter_2_DB"(Y17_RotCilipozDesno := "dbDigitalValves".Y17_RotCilipozDesno,
	                      Y18_RotCilipozLevo := "dbDigitalValves".Y18_RotCilipozLevo,
	                      Y6_DrcaLocev_Des := "dbDigitalValves".Y6_DrcaLocev_Des,
	                      Y7_DrcaLocev_Lev := "dbDigitalValves".Y7_DrcaLocev_Lev);
	
	"op_ButtonHelix_3_DB"(SEMAFOR_ZELENA:= "dbDigitalValves".SEMAFOR_ZELENA,
	                      SEMAFOR_RUMENA:= "dbDigitalValves".SEMAFOR_RUMENA,
	                      SEMAFOR_RDECA:= "dbDigitalValves".SEMAFOR_RDECA,
	                      VKLOP_VIBRATORJA:= "dbMotors".VKLOP_VIBRATORJA,
	                      VKLOP_M_TRACNEGA_TRANS_NOGIC:= "dbMotors".VKLOP_M_TRACNEGA_TRANS_NOGIC);
	
END_FUNCTION

FUNCTION "fcUtilities" : Void
{ S7_Optimized_Access := 'FALSE' }
VERSION : 0.1
   VAR_TEMP 
      i : Int;
   END_VAR

   VAR CONSTANT 
      LightPulseTime : Int := 20;
      LightPauseTime : Int := 10;
   END_VAR


BEGIN
	// Short summary:
	(*
	  Function that stores functionality that is not part of phases, but 
	  needed for normal operation
	*)
	// 
	//**********************************************************************
	// Revision control:
	//----------------------------------------------------------------------
	// Use only for revisions of original code
	// V0.01
	// Description of revision
	
	
	//----------------------------------------------------------------------
	// Comments:
	(*
	  Every change in the code is documented with following:
	  // CCC-yyymmdd: .....
	  yyyy year when change was made
	  mm   month when change was made
	  dd   day when change was made
	  CCC  authors initials
	*)
	
	// ************* BEGIN - Indication lights ************* //
	// ***** GREEN ***** //
	"dbTimers".Num[12].PRE := #LightPulseTime;
	"dbTimers".Num[16].PRE := #LightPauseTime;
	"dbTimers".Num[12].EE := ("dbUnit".Unit[1].StartStop) AND NOT "dbUtilities".GreenLightFlashFlag;
	"dbTimers".Num[16].EE := ("dbUnit".Unit[1].StartStop) AND "dbUtilities".GreenLightFlashFlag;
	
	IF "dbTimers".Num[12].EE AND "dbTimers".Num[12].DN THEN
	    "dbUtilities".GreenLightFlashFlag := 1; 
	ELSIF "dbTimers".Num[16].EE AND "dbTimers".Num[16].DN THEN
	    "dbUtilities".GreenLightFlashFlag := 0;
	END_IF;
	// GREEN LIGHT FLASHING or GREEN ALWAYS ON
	IF ("dbTimers".Num[12].EE AND "dbTimers".Num[12].TT) // FLASHING- ready for run
	THEN
	  ; // "dbDigitalValves".SEMAFOR_ZELENA.AutoON := True;
	END_IF;
	"dbDigitalValves".SEMAFOR_ZELENA.AutoON := ("dbUnit".Unit[1].StartStop);
	// ***** GREEN ***** //
	
	// ***** RED ***** //
	"dbTimers".Num[20].PRE := #LightPulseTime;
	"dbTimers".Num[24].PRE := #LightPauseTime;
	"dbTimers".Num[20].EE := "dbUnit".Unit[1].AlarmsPresent AND NOT "dbUtilities".RedLightFlashFlag;
	"dbTimers".Num[24].EE := "dbUnit".Unit[1].AlarmsPresent AND "dbUtilities".RedLightFlashFlag;
	
	IF "dbTimers".Num[20].EE AND "dbTimers".Num[20].DN THEN
	    "dbUtilities".RedLightFlashFlag := 1;
	ELSIF "dbTimers".Num[24].EE AND "dbTimers".Num[24].DN THEN
	    "dbUtilities".RedLightFlashFlag := 0;
	END_IF;
	
	// RED LIGHT FLASHING or RED ALWAYS ON
	IF ("dbTimers".Num[20].EE AND "dbTimers".Num[20].TT) THEN // FLASHING
	  "dbDigitalValves".SEMAFOR_RDECA.AutoON := True;
	END_IF;
	// ***** RED ***** //
	
	// ***** YELLOW ***** //
	"dbTimers".Num[28].PRE := #LightPulseTime;
	"dbTimers".Num[32].PRE := #LightPauseTime;
	(* 20210517_PRA
	"dbTimers".Num[28].EE := "ph_Helix_1_DB".CurrentStep=10 AND "ph_Helix_1_DB".InsertNewButtom>0
	                          AND NOT "dbUtilities".YellowLightFlashFlag;
	"dbTimers".Num[32].EE :=  "ph_Helix_1_DB".CurrentStep=10 AND "ph_Helix_1_DB".InsertNewButtom>0
	                          AND "dbUtilities".YellowLightFlashFlag;
	*)
	"dbTimers".Num[28].EE := (("ph_Helix_1_DB".CurrentStep=10 AND "ph_Helix_1_DB".InsertNewButtom>0) OR "dbAlarms".PLI[3, 8])
	                          AND NOT "dbUtilities".YellowLightFlashFlag;
	"dbTimers".Num[32].EE :=  (("ph_Helix_1_DB".CurrentStep=10 AND "ph_Helix_1_DB".InsertNewButtom>0) OR "dbAlarms".PLI[3, 8])
	                          AND "dbUtilities".YellowLightFlashFlag;
	
	IF "dbTimers".Num[28].EE AND "dbTimers".Num[28].DN THEN
	    "dbUtilities".YellowLightFlashFlag := 1;
	ELSIF "dbTimers".Num[32].EE AND "dbTimers".Num[32].DN THEN
	    "dbUtilities".YellowLightFlashFlag := 0;
	END_IF;
	// YELLOW LIGHT FLASHING or GREEN ALWAYS ON
	IF ("dbTimers".Num[28].EE AND "dbTimers".Num[28].TT) // FLASHING
	THEN
	  "dbDigitalValves".SEMAFOR_RUMENA.AutoON := True;
	END_IF;
	// ***** YELLOW ***** //
	
	// ************* END - Indication lights ************* //
	
	// ************* BEIN - User logged out ************* //
	IF "dbHMIUser".UserLoggOffTime > 59 THEN
	    "dbHMIUser".UserLoggOffTime := 58;
	END_IF;
	IF ("dbHMIUser".PLCUserLogOut=0) AND ("dbHMIUser".PLCUserLogOut_OLD=1) THEN            
	    "dbHMIUser".CurrentUsername := '';
	END_IF;
	    
	"dbTimers".Num[4].PRE := "dbHMIUser".UserLoggOffTime * 60 * 10; // 100 msec
	"dbTimers".Num[4].EE := "dbHMIUser".CurrUser_LEN > 0;
	IF "dbHMIUser".CurrUser_LEN > 0 THEN
	    "dbHMIUser".PLCUserLogOut := 1;
	END_IF;
	"dbTimers".Num[4].RS := "dbUnit".Unit[1].StartStop;
	IF "FirstScan" THEN
	    "dbHMIUser".CurrentUsername := '';
	END_IF;
	IF "dbTimers".Num[4].EE AND "dbTimers".Num[4].DN THEN            
	    "dbHMIUser".PLCUserLogOut := 0;
	    "dbHMIUser".CurrentUsername := '';
	END_IF;
	
	"dbHMIUser".CurrUser_LEN := LEN("dbHMIUser".CurrentUsername); // if 0 user not logged IN, if > 0 user is logged IN
	"dbHMIUser".PLCUserLogOut_OLD := "dbHMIUser".PLCUserLogOut;
	// ************* END - User logged out ************* //
	
